(* IEC 61131-3 sources: beckhoffAutomationInterface/ST/Shark/Lib/Sequences, 14 files *)

(* ---- GVL_SequenceConstants.st ---- *)
(* Constants used by Lib/Sequences/* function blocks.
   Lifted from App-side GVL_Constants so Lib code does not depend on
   App-scoped configuration.

   These describe properties of the shared hardware (Bronkhorst PCV needle
   valve) and are identical across all machines that use this valve. *)
{attribute 'qualified_only'}
VAR_GLOBAL CONSTANT
    // Pressure Control Valve (PCV / Needle Valve) Setpoints
    // Bronkhorst Modbus needle valve: 0.0 bar = fully open, 3.0 bar = fully closed
    PCV_CLOSED_SETPOINT : LREAL := 3.0;     // Setpoint that fully closes needle valve (no flow)
    PCV_OPEN_SETPOINT   : LREAL := 0.0;     // Setpoint that fully opens needle valve (max flow)
END_VAR

(* ---- FB_BubblerLeakTestSequence.st ---- *)
(*
FB_BubblerLeakTestSequence
Pressurizes the manifold through a specific bubbler, seals it, and monitors
pressure drop over a configurable test duration.

SEQUENCE:
  1. GasStop:     Ensure both sides shut down
  2. Pressurize:  Fill manifold via MFC + bubbler (CM -> HM path)
  3. Seal:        Close all valves, zero MFC
  4. Stabilize:   Wait for pressure to equalize
  5. Test:        Monitor pressure drop over testDuration
  6. Analyze:     Compare drop vs threshold
  7. Cleanup:     Close all valves
  8. Complete:    Report results

HARDWARE:
  - Side MFC + gas iso valve (carrier gas)
  - CM bubbler valve + CM purge valve (fill path)
  - HM bubbler valve + HM purge valve (propagation to HM)
  - CM/HM pressure sensors (monitor)

OUTPUT:
  - bLeakDetected, fColdManifoldPressureDrop, fHotManifoldPressureDrop
*)
FUNCTION_BLOCK FB_BubblerLeakTestSequence IMPLEMENTS I_TreeNode
VAR
    // Internal State
    _bInitialized    : BOOL := FALSE;
    _bParamsConfigured : BOOL := FALSE;
    _ePhase          : INT := 0;

    // Hardware References
    _ipGasIsoValve        : I_Valve;
    _ipCMBubblerValve     : I_Valve;
    _ipHMBubblerValve     : I_Valve;
    _ipCMPurgeValve       : I_Valve;
    _ipHMPurgeValve       : I_Valve;
    _ipCMVacuumIsoValve   : I_Valve;
    _ipHMVacuumIsoValve   : I_Valve;
    _ipCMPressureSensor   : I_Sensor;
    _ipHMPressureSensor   : I_Sensor;
    _ipMFCController      : I_Controller;

    // Gas stop
    _fbGasStop            : FB_GasStopSequence;

    // Parameters
    _stParams             : ST_CmdBubblerLeakTest;
    _eSide                : E_GasSide;

    // Measurement
    _rCMPressureInitial   : LREAL;
    _rHMPressureInitial   : LREAL;
    _rCMPressureFinal     : LREAL;
    _rHMPressureFinal     : LREAL;

    // Timing
    _fbTimer              : TON;

    // Status
    _bError               : BOOL;
    _sErrorMsg            : STRING(255);
END_VAR

// Output results (readable after completion)
VAR_OUTPUT
    bLeakDetected             : BOOL;
    bColdManifoldLeak         : BOOL;
    bHotManifoldLeak          : BOOL;
    fColdManifoldPressureDrop : LREAL;
    fHotManifoldPressureDrop  : LREAL;
    fPressureDrop             : LREAL;     // max of CM/HM
END_VAR

VAR CONSTANT
    PHASE_IDLE       : INT := 0;
    PHASE_GAS_STOP   : INT := 1;
    PHASE_FILL       : INT := 2;
    PHASE_SEAL       : INT := 3;
    PHASE_STABILIZE  : INT := 4;
    PHASE_TEST       : INT := 5;
    PHASE_ANALYZE    : INT := 6;
    PHASE_CLEANUP    : INT := 7;
    PHASE_DONE       : INT := 8;
    PHASE_ERROR      : INT := 99;
END_VAR

METHOD PUBLIC Init : BOOL
VAR_INPUT
    ipProvider    : I_HardwareProvider;
    eSide         : E_GasSide;
    nBubblerIndex : DINT;
END_VAR
    _bInitialized := FALSE;
    _bParamsConfigured := FALSE;
    _ePhase := PHASE_IDLE;
    _bError := FALSE;
    _sErrorMsg := '';
    _eSide := eSide;

    IF ipProvider = 0 THEN
        GVL_ErrorLogger.Logger.LogError('FB_BubblerLeakTestSequence', E_ErrorId.ERR_GEN_NULL_POINTER, 'Provider is null');
        RETURN;
    END_IF

    IF NOT _fbGasStop.Init(ipProvider := ipProvider, eSide := eSide) THEN RETURN; END_IF

    _ipGasIsoValve := ipProvider.GetGasIsoValve(eSide, nBubblerIndex);
    _ipCMBubblerValve := ipProvider.GetCMBubblerValve(eSide, nBubblerIndex);
    _ipHMBubblerValve := ipProvider.GetHMBubblerValve(eSide, nBubblerIndex);
    _ipCMPurgeValve := ipProvider.GetCMPurgeValve(eSide);
    _ipHMPurgeValve := ipProvider.GetHMPurgeValve(eSide);
    _ipCMVacuumIsoValve := ipProvider.GetCMVacuumIsoValve(eSide);
    _ipHMVacuumIsoValve := ipProvider.GetHMVacuumIsoValve(eSide);
    _ipCMPressureSensor := ipProvider.GetCMPressureSensor(eSide);
    _ipHMPressureSensor := ipProvider.GetHMPressureSensor(eSide);
    _ipMFCController := ipProvider.GetMFCController(eSide);

    IF _ipGasIsoValve = 0 OR _ipCMBubblerValve = 0 OR _ipHMBubblerValve = 0 OR
       _ipCMPurgeValve = 0 OR _ipHMPurgeValve = 0 OR
       _ipCMPressureSensor = 0 OR _ipHMPressureSensor = 0 OR _ipMFCController = 0 THEN
        GVL_ErrorLogger.Logger.LogError('FB_BubblerLeakTestSequence', E_ErrorId.ERR_GEN_NULL_POINTER, 'One or more hardware references are null');
        RETURN;
    END_IF

    _bInitialized := TRUE;
    Init := TRUE;
END_METHOD

METHOD PUBLIC SetParams
VAR_INPUT
    stParams : ST_CmdBubblerLeakTest;
END_VAR
    IF NOT _bInitialized THEN RETURN; END_IF
    _stParams := stParams;
    _bParamsConfigured := TRUE;
END_METHOD

METHOD PUBLIC Tick : ST_NodeResult
VAR
    stResult : ST_NodeResult;
END_VAR
    IF NOT _bInitialized THEN
        Tick.eStatus := E_NodeStatus.FAILURE;
        Tick.bHasError := TRUE;
        Tick.stError.eErrorId := E_ErrorId.ERR_GEN_INITIALIZATION;
        Tick.stError.sSource := 'FB_BubblerLeakTestSequence';
        Tick.stError.sMessage := 'Init must be called before Tick';
        Tick.sDescription := Tick.stError.sMessage;
        RETURN;
    END_IF

    IF NOT _bParamsConfigured THEN
        Tick.eStatus := E_NodeStatus.FAILURE;
        Tick.bHasError := TRUE;
        Tick.stError.eErrorId := E_ErrorId.ERR_GEN_NOT_CONFIGURED;
        Tick.stError.sSource := 'FB_BubblerLeakTestSequence';
        Tick.stError.sMessage := 'SetParams must be called before Tick';
        Tick.sDescription := Tick.stError.sMessage;
        RETURN;
    END_IF

    CASE _ePhase OF
        PHASE_IDLE:
            // Reset outputs
            bLeakDetected := FALSE;
            bColdManifoldLeak := FALSE;
            bHotManifoldLeak := FALSE;
            fColdManifoldPressureDrop := 0.0;
            fHotManifoldPressureDrop := 0.0;
            fPressureDrop := 0.0;
            _fbGasStop.Reset();
            _ePhase := PHASE_GAS_STOP;

        PHASE_GAS_STOP:
            stResult := _fbGasStop.Tick();
            IF stResult.eStatus = E_NodeStatus.SUCCESS THEN
                _ePhase := PHASE_FILL;
                _fbTimer(IN := FALSE);
            ELSIF stResult.eStatus = E_NodeStatus.FAILURE THEN
                _SetError('Gas stop failed');
            END_IF

        PHASE_FILL:
            // Open path: GasIso -> CMBubbler -> CMPurge -> HMPurge -> HMBubbler
            // Set MFC to test flow, wait for fill pressure
            IF NOT _fbTimer.IN THEN
                _ipMFCController.SetSetpoint(REAL_TO_LREAL(_stParams.testFlowRate));
                _ipGasIsoValve.Open();
                _ipCMBubblerValve.Open();
                _ipCMPurgeValve.Open();
                _ipHMPurgeValve.Open();
                _ipHMBubblerValve.Open();
                // Close exhaust paths
                IF _ipCMVacuumIsoValve <> 0 THEN _ipCMVacuumIsoValve.Close(); END_IF
                IF _ipHMVacuumIsoValve <> 0 THEN _ipHMVacuumIsoValve.Close(); END_IF
            END_IF
            _fbTimer(IN := TRUE, PT := DINT_TO_TIME(_stParams.pressureTimeout));
            IF _ipCMPressureSensor.GetMeasurement() >= REAL_TO_LREAL(_stParams.fillPressure) AND
               _ipHMPressureSensor.GetMeasurement() >= REAL_TO_LREAL(_stParams.fillPressure) THEN
                _ePhase := PHASE_SEAL;
                _fbTimer(IN := FALSE);
            ELSIF _fbTimer.Q THEN
                _SetError('Timeout waiting for fill pressure');
            END_IF

        PHASE_SEAL:
            // Close everything, zero MFC
            _ipMFCController.SetSetpoint(0.0);
            _ipGasIsoValve.Close();
            _ipCMBubblerValve.Close();
            _ipHMBubblerValve.Close();
            _ipCMPurgeValve.Close();
            _ipHMPurgeValve.Close();
            _fbTimer(IN := FALSE);
            _ePhase := PHASE_STABILIZE;

        PHASE_STABILIZE:
            _fbTimer(IN := TRUE, PT := DINT_TO_TIME(_stParams.stabilizationTime));
            IF _fbTimer.Q THEN
                // Record initial pressures
                _rCMPressureInitial := _ipCMPressureSensor.GetMeasurement();
                _rHMPressureInitial := _ipHMPressureSensor.GetMeasurement();
                _fbTimer(IN := FALSE);
                _ePhase := PHASE_TEST;
            END_IF

        PHASE_TEST:
            _fbTimer(IN := TRUE, PT := DINT_TO_TIME(_stParams.testDuration));
            IF _fbTimer.Q THEN
                // Record final pressures
                _rCMPressureFinal := _ipCMPressureSensor.GetMeasurement();
                _rHMPressureFinal := _ipHMPressureSensor.GetMeasurement();
                _fbTimer(IN := FALSE);
                _ePhase := PHASE_ANALYZE;
            END_IF

        PHASE_ANALYZE:
            // Calculate pressure drops
            fColdManifoldPressureDrop := _rCMPressureInitial - _rCMPressureFinal;
            fHotManifoldPressureDrop := _rHMPressureInitial - _rHMPressureFinal;

            bColdManifoldLeak := (fColdManifoldPressureDrop > REAL_TO_LREAL(_stParams.leakThreshold));
            bHotManifoldLeak := (fHotManifoldPressureDrop > REAL_TO_LREAL(_stParams.leakThreshold));
            bLeakDetected := bColdManifoldLeak OR bHotManifoldLeak;

            // Max drop for summary
            IF fColdManifoldPressureDrop > fHotManifoldPressureDrop THEN
                fPressureDrop := fColdManifoldPressureDrop;
            ELSE
                fPressureDrop := fHotManifoldPressureDrop;
            END_IF

            _ePhase := PHASE_CLEANUP;

        PHASE_CLEANUP:
            // Ensure all valves closed
            _ipCMBubblerValve.Close();
            _ipHMBubblerValve.Close();
            _ipCMPurgeValve.Close();
            _ipHMPurgeValve.Close();
            _ipGasIsoValve.Close();
            _ePhase := PHASE_DONE;

        PHASE_DONE:
            // Stay done

        PHASE_ERROR:
            // Stay in error
    END_CASE

    IF _ePhase = PHASE_DONE THEN
        Tick.eStatus := E_NodeStatus.SUCCESS;
        Tick.rProgress := 100.0;
        IF bLeakDetected THEN
            Tick.sDescription := CONCAT('LEAK DETECTED - Drop: ', LREAL_TO_STRING(fPressureDrop));
        ELSE
            Tick.sDescription := 'Leak test PASSED';
        END_IF
    ELSIF _ePhase = PHASE_ERROR THEN
        Tick.eStatus := E_NodeStatus.FAILURE;
        Tick.bHasError := TRUE;
        Tick.stError.eErrorId := E_ErrorId.ERR_GEN_INTERNAL;
        Tick.stError.sSource := 'FB_BubblerLeakTestSequence';
        Tick.stError.sMessage := _sErrorMsg;
        Tick.sDescription := _sErrorMsg;
    ELSE
        Tick.eStatus := E_NodeStatus.RUNNING;
        Tick.sDescription := CONCAT('Leak Test: Phase ', INT_TO_STRING(_ePhase));
    END_IF
END_METHOD

METHOD PRIVATE _SetError
VAR_INPUT
    sMsg : STRING(255);
END_VAR
    _sErrorMsg := sMsg;
    _bError := TRUE;
    _ePhase := PHASE_ERROR;
END_METHOD

METHOD PUBLIC Reset : BOOL
    _ePhase := PHASE_IDLE;
    _bError := FALSE;
    _sErrorMsg := '';
    _fbTimer(IN := FALSE);
    bLeakDetected := FALSE;
    bColdManifoldLeak := FALSE;
    bHotManifoldLeak := FALSE;
    fColdManifoldPressureDrop := 0.0;
    fHotManifoldPressureDrop := 0.0;
    fPressureDrop := 0.0;
    _fbGasStop.Reset();
    Reset := TRUE;
END_METHOD

METHOD PUBLIC Halt
    IF _ipMFCController <> 0 THEN _ipMFCController.SetSetpoint(0.0); END_IF
    IF _ipGasIsoValve <> 0 THEN _ipGasIsoValve.Close(); END_IF
    IF _ipCMBubblerValve <> 0 THEN _ipCMBubblerValve.Close(); END_IF
    IF _ipHMBubblerValve <> 0 THEN _ipHMBubblerValve.Close(); END_IF
    IF _ipCMPurgeValve <> 0 THEN _ipCMPurgeValve.Close(); END_IF
    IF _ipHMPurgeValve <> 0 THEN _ipHMPurgeValve.Close(); END_IF
    Reset();
END_METHOD

PROPERTY PUBLIC NodeName : STRING(50)
    GET
        NodeName := 'BubblerLeakTest';
    END_GET
END_PROPERTY

END_FUNCTION_BLOCK

(* ---- FB_BubblerPurgeSequence.st ---- *)
(*
FB_BubblerPurgeSequence
Purge a specific bubbler: Prepare exhaust -> CM purge -> delay -> HM purge.
*)
FUNCTION_BLOCK FB_BubblerPurgeSequence IMPLEMENTS I_TreeNode
VAR
    _seq : FB_SequenceNode;
    // Steps
    stepPrepareExhaust : FB_PrepareExhaustSequence;
    stepBubblerPurgeCM : FB_BubblerPurgeCMSequence;
    stepDelay          : FB_WaitNode;
    stepBubblerPurgeHM : FB_BubblerPurgeHMSequence;

    // Internal state
    _bInitialized    : BOOL := FALSE;
    _eSide           : E_GasSide;
    _nBubblerIndex   : DINT;
END_VAR

VAR CONSTANT
    SWITCH_DELAY : TIME := T#2S;
END_VAR

METHOD PUBLIC Init : BOOL
VAR_INPUT
    ipProvider    : I_HardwareProvider;
    eSide         : E_GasSide;
    nBubblerIndex : DINT;
END_VAR
    IF _bInitialized THEN
        IF _eSide = eSide AND _nBubblerIndex = nBubblerIndex THEN
            Init := TRUE;
            RETURN;
        END_IF
        _seq.ClearChildren();
        _bInitialized := FALSE;
    END_IF

    IF ipProvider = 0 THEN
        GVL_ErrorLogger.Logger.LogError('FB_BubblerPurgeSequence', E_ErrorId.ERR_GEN_NULL_POINTER, 'Provider is null');
        RETURN;
    END_IF
    _eSide := eSide;
    _nBubblerIndex := nBubblerIndex;

    stepPrepareExhaust.Init(ipProvider, eSide);
    stepPrepareExhaust.NodeName := 'PrepareExhaust';
    _seq.AddChild(stepPrepareExhaust);

    stepBubblerPurgeCM.Init(ipProvider, eSide, nBubblerIndex);
    stepBubblerPurgeCM.NodeName := 'BubblerPurgeCM';
    _seq.AddChild(stepBubblerPurgeCM);

    stepDelay.Init(tWaitTime := SWITCH_DELAY, sNodeName := 'SwitchDelay');
    _seq.AddChild(stepDelay);

    stepBubblerPurgeHM.Init(ipProvider, eSide, nBubblerIndex);
    stepBubblerPurgeHM.NodeName := 'BubblerPurgeHM';
    _seq.AddChild(stepBubblerPurgeHM);

    _seq.sName := CONCAT(CONCAT('BubblerPurgeFull_Side', TO_STRING(eSide)), CONCAT('_Idx', TO_STRING(nBubblerIndex)));

    _bInitialized := TRUE;
    Init := TRUE;
END_METHOD

METHOD PUBLIC SetParams
VAR_INPUT
    stCmd : ST_CmdPurge;
END_VAR
    IF NOT _bInitialized THEN RETURN; END_IF

    stepBubblerPurgeCM.SetParams(
        nPurgeCycles           := stCmd.coldManifoldPurgeCycles,
        rPurgeFlowRate         := REAL_TO_LREAL(stCmd.purgeGasFlow),
        rPurgePressure         := REAL_TO_LREAL(stCmd.purgeHighPressureLimit),
        rEvacuationPressure    := REAL_TO_LREAL(stCmd.purgeLowPressureLimit),
        tPressurizationTimeout := DINT_TO_TIME(stCmd.highPressureTimeout),
        tEvacuationTimeout     := DINT_TO_TIME(stCmd.lowPressureTimeout)
    );

    stepBubblerPurgeHM.SetParams(
        nPurgeCycles           := stCmd.hotManifoldPurgeCycles,
        rPurgeFlowRate         := REAL_TO_LREAL(stCmd.purgeGasFlow),
        rPurgePressure         := REAL_TO_LREAL(stCmd.purgeHighPressureLimit),
        rFinalPressure         := REAL_TO_LREAL(stCmd.hotManifoldOperatingPressure),
        rEvacuationPressure    := REAL_TO_LREAL(stCmd.purgeLowPressureLimit),
        tPressurizationTimeout := DINT_TO_TIME(stCmd.highPressureTimeout),
        tEvacuationTimeout     := DINT_TO_TIME(stCmd.lowPressureTimeout)
    );
END_METHOD

PROPERTY PUBLIC NodeName : STRING(50)
    GET
        NodeName := _seq.sName;
    END_GET
    SET
        _seq.sName := NodeName;
    END_SET
END_PROPERTY

METHOD Tick : ST_NodeResult
    IF NOT _bInitialized THEN
        Tick.eStatus := E_NodeStatus.FAILURE;
        Tick.bHasError := TRUE;
        Tick.stError.eErrorId := E_ErrorId.ERR_GEN_INITIALIZATION;
        Tick.stError.sSource := 'FB_BubblerPurgeSequence';
        Tick.stError.sMessage := 'Init must be called before Tick';
        Tick.sDescription := Tick.stError.sMessage;
        RETURN;
    END_IF

    Tick := _seq.Tick();
END_METHOD

{attribute 'estimated-stack-usage' := '500'}
METHOD Reset : BOOL
    Reset := _seq.Reset();
END_METHOD

{attribute 'estimated-stack-usage' := '500'}
METHOD Halt
    _seq.Halt();
END_METHOD

END_FUNCTION_BLOCK

(* ---- FB_ChuckVacuumHoldSequence.st ---- *)
// FB_ChuckVacuumHoldSequence (Lib)
//
// Machine-agnostic chuck-vacuum hold sequence. All hardware-specific
// behavior (pump topology, vent valve presence, sensor type) is delegated
// to the machine-specific I_ChuckVacuumSystem implementation provided by
// the hardware provider.
//
// SEQUENCE:
//   Idle           -> PrepareForHold() then wait pump stabilize
//   VerifyingPump  -> after stabilize, open zone valves
//   OpeningValves  -> hierarchical open 1..nZoneCount, then watch sensor
//   WaitingVacuum  -> until IsVacuumHeld OR timeout
//   Done / Error
FUNCTION_BLOCK FB_ChuckVacuumHoldSequence IMPLEMENTS I_TreeNode
VAR
    _bInitialized    : BOOL := FALSE;
    _eState          : E_ChuckVacuumState := E_ChuckVacuumState.Idle;

    _ipChuckVacuum   : I_ChuckVacuumSystem;

    // Parameters
    _nZoneCount              : INT  := 1;
    _tTimeout                : TIME := T#1M;
    _rLockPressureThreshold  : LREAL := 0.65;

    _fbTimer         : TON;
    _bError          : BOOL;
    _sErrorMsg       : STRING(255);
END_VAR

VAR CONSTANT
    PUMP_STABILIZE_TIME : TIME := T#500MS;
END_VAR

METHOD PUBLIC Init : BOOL
VAR_INPUT
    ipProvider : I_HardwareProvider;
END_VAR
    _bInitialized := FALSE;
    _eState := E_ChuckVacuumState.Idle;
    _bError := FALSE;
    _sErrorMsg := '';

    IF ipProvider = 0 THEN
        GVL_ErrorLogger.Logger.LogError('FB_ChuckVacuumHoldSequence', E_ErrorId.ERR_GEN_NULL_POINTER, 'Provider is null');
        RETURN;
    END_IF

    _ipChuckVacuum := ipProvider.GetChuckVacuumSystem();
    IF _ipChuckVacuum = 0 THEN
        GVL_ErrorLogger.Logger.LogError('FB_ChuckVacuumHoldSequence', E_ErrorId.ERR_GEN_NULL_POINTER, 'Chuck vacuum subsystem not available');
        RETURN;
    END_IF

    IF NOT _ipChuckVacuum.IsInitialized() THEN
        GVL_ErrorLogger.Logger.LogError('FB_ChuckVacuumHoldSequence', E_ErrorId.ERR_GEN_NULL_POINTER, 'Chuck vacuum subsystem not initialized');
        RETURN;
    END_IF

    _bInitialized := TRUE;
    Init := TRUE;
END_METHOD

METHOD PUBLIC SetParams
VAR_INPUT
    stParams : ST_ChuckVacuumHold;
END_VAR
VAR
    nMax : INT;
END_VAR
    IF NOT _bInitialized THEN RETURN; END_IF
    nMax := _ipChuckVacuum.GetMaxZoneCount();
    _nZoneCount := LIMIT(1, stParams.iSelectZone, nMax);
    _tTimeout := stParams.tPressureTimeout;
    _rLockPressureThreshold := REAL_TO_LREAL(stParams.fLockPressureThreshold);
END_METHOD

METHOD PUBLIC Tick : ST_NodeResult
VAR
    i : INT;
END_VAR
    IF NOT _bInitialized THEN
        _sErrorMsg := 'Init must be called before Tick';
        _bError := TRUE;
        _eState := E_ChuckVacuumState.Error;
        Tick.eStatus := E_NodeStatus.FAILURE;
        Tick.bHasError := TRUE;
        Tick.stError.eErrorId := E_ErrorId.ERR_GEN_INITIALIZATION;
        Tick.stError.sSource := 'FB_ChuckVacuumHoldSequence';
        Tick.stError.sMessage := _sErrorMsg;
        Tick.sDescription := _sErrorMsg;
        RETURN;
    END_IF

    CASE _eState OF
        E_ChuckVacuumState.Idle:
            // Close vent (if any), ensure pump source is active
            _ipChuckVacuum.PrepareForHold();
            _eState := E_ChuckVacuumState.VerifyingPump;
            _fbTimer(IN := FALSE);

        E_ChuckVacuumState.VerifyingPump:
            // Brief stabilization window for pump/vent valve to settle
            _fbTimer(IN := TRUE, PT := PUMP_STABILIZE_TIME);
            IF _fbTimer.Q THEN
                _fbTimer(IN := FALSE);
                _eState := E_ChuckVacuumState.OpeningValves;
            END_IF

        E_ChuckVacuumState.OpeningValves:
            // Open zone valves hierarchically (innermost first)
            FOR i := 1 TO _nZoneCount DO
                _ipChuckVacuum.OpenZone(nZone := i);
            END_FOR
            _eState := E_ChuckVacuumState.WaitingVacuum;
            _fbTimer(IN := FALSE);

        E_ChuckVacuumState.WaitingVacuum:
            _fbTimer(IN := TRUE, PT := _tTimeout);
            IF _fbTimer.Q THEN
                _sErrorMsg := 'Timeout waiting for vacuum';
                _bError := TRUE;
                _eState := E_ChuckVacuumState.Error;
            ELSIF _ipChuckVacuum.IsVacuumHeld(nActiveZoneCount := _nZoneCount, rThreshold := _rLockPressureThreshold) THEN
                _eState := E_ChuckVacuumState.Done;
            END_IF

        E_ChuckVacuumState.Done:
            ; // terminal
        E_ChuckVacuumState.Error:
            ; // terminal until Reset
    END_CASE

    Tick.eStatus := E_NodeStatus.RUNNING;
    Tick.rProgress := 0.0;
    Tick.bHasError := _bError;
    Tick.sDescription := 'Applying Vacuum';

    IF _eState = E_ChuckVacuumState.Done THEN
        Tick.eStatus := E_NodeStatus.SUCCESS;
        Tick.rProgress := 100.0;
        Tick.sDescription := 'Vacuum Held';
    ELSIF _eState = E_ChuckVacuumState.Error THEN
        Tick.eStatus := E_NodeStatus.FAILURE;
        Tick.bHasError := TRUE;
        Tick.stError.eErrorId := E_ErrorId.ERR_GEN_TIMEOUT;
        Tick.stError.sSource := 'FB_ChuckVacuumHoldSequence';
        Tick.stError.sMessage := _sErrorMsg;
        Tick.stError.fExpectedValue := TO_REAL(_rLockPressureThreshold);
        Tick.stError.sUnits := 'bar';
        Tick.sDescription := _sErrorMsg;
    END_IF
END_METHOD

METHOD PUBLIC GetState : E_ChuckVacuumState
    GetState := _eState;
END_METHOD

METHOD PUBLIC Reset : BOOL
    _eState := E_ChuckVacuumState.Idle;
    _bError := FALSE;
    _sErrorMsg := '';
    _fbTimer(IN := FALSE);
    IF _ipChuckVacuum <> 0 THEN
        _ipChuckVacuum.Reset();
    END_IF
    Reset := TRUE;
END_METHOD

METHOD PUBLIC Halt
    Reset();
END_METHOD

END_FUNCTION_BLOCK

(* ---- FB_ChuckVacuumReleaseSequence.st ---- *)
// FB_ChuckVacuumReleaseSequence (Lib)
//
// Machine-agnostic chuck-vacuum release sequence. All hardware-specific
// behavior is delegated to the I_ChuckVacuumSystem implementation.
//
// SEQUENCE:
//   Idle           -> close all zones, BeginRelease()  (opens vent if any)
//   WaitingVacuum  -> until IsVacuumReleased OR timeout
//   On release    -> FinishRelease() (stops pump if dedicated)
//   Done / Error
FUNCTION_BLOCK FB_ChuckVacuumReleaseSequence IMPLEMENTS I_TreeNode
VAR
    _bInitialized    : BOOL := FALSE;
    _eState          : E_ChuckVacuumState := E_ChuckVacuumState.Idle;

    _ipChuckVacuum   : I_ChuckVacuumSystem;

    // Parameters
    _tTimeout                   : TIME  := T#1M;
    _rReleasePressureThreshold  : LREAL := 0.8;

    _fbTimer         : TON;
    _bError          : BOOL;
    _sErrorMsg       : STRING(255);
END_VAR

METHOD PUBLIC Init : BOOL
VAR_INPUT
    ipProvider : I_HardwareProvider;
END_VAR
    _bInitialized := FALSE;
    _eState := E_ChuckVacuumState.Idle;
    _bError := FALSE;
    _sErrorMsg := '';

    IF ipProvider = 0 THEN
        GVL_ErrorLogger.Logger.LogError('FB_ChuckVacuumReleaseSequence', E_ErrorId.ERR_GEN_NULL_POINTER, 'Provider is null');
        RETURN;
    END_IF

    _ipChuckVacuum := ipProvider.GetChuckVacuumSystem();
    IF _ipChuckVacuum = 0 THEN
        GVL_ErrorLogger.Logger.LogError('FB_ChuckVacuumReleaseSequence', E_ErrorId.ERR_GEN_NULL_POINTER, 'Chuck vacuum subsystem not available');
        RETURN;
    END_IF

    IF NOT _ipChuckVacuum.IsInitialized() THEN
        GVL_ErrorLogger.Logger.LogError('FB_ChuckVacuumReleaseSequence', E_ErrorId.ERR_GEN_NULL_POINTER, 'Chuck vacuum subsystem not initialized');
        RETURN;
    END_IF

    _bInitialized := TRUE;
    Init := TRUE;
END_METHOD

METHOD PUBLIC SetParams
VAR_INPUT
    stParams : ST_ChuckVacuumRelease;
END_VAR
    IF NOT _bInitialized THEN RETURN; END_IF
    _tTimeout := stParams.tPressureTimeout;
    _rReleasePressureThreshold := REAL_TO_LREAL(stParams.fReleasePressureThreshold);
END_METHOD

METHOD PUBLIC Tick : ST_NodeResult
VAR
    i, nMax : INT;
END_VAR
    IF NOT _bInitialized THEN
        _sErrorMsg := 'Init must be called before Tick';
        _bError := TRUE;
        _eState := E_ChuckVacuumState.Error;
        Tick.eStatus := E_NodeStatus.FAILURE;
        Tick.bHasError := TRUE;
        Tick.stError.eErrorId := E_ErrorId.ERR_GEN_INITIALIZATION;
        Tick.stError.sSource := 'FB_ChuckVacuumReleaseSequence';
        Tick.stError.sMessage := _sErrorMsg;
        Tick.sDescription := _sErrorMsg;
        RETURN;
    END_IF

    CASE _eState OF
        E_ChuckVacuumState.Idle:
            _eState := E_ChuckVacuumState.OpeningValves;
            _fbTimer(IN := FALSE);

        E_ChuckVacuumState.OpeningValves:
            // Close every zone, then open vent (if any) via BeginRelease
            nMax := _ipChuckVacuum.GetMaxZoneCount();
            FOR i := 1 TO nMax DO
                _ipChuckVacuum.CloseZone(nZone := i);
            END_FOR
            _ipChuckVacuum.BeginRelease();
            _eState := E_ChuckVacuumState.WaitingVacuum;
            _fbTimer(IN := FALSE);

        E_ChuckVacuumState.WaitingVacuum:
            _fbTimer(IN := TRUE, PT := _tTimeout);
            IF _fbTimer.Q THEN
                _sErrorMsg := 'Timeout waiting for vacuum release';
                _bError := TRUE;
                _eState := E_ChuckVacuumState.Error;
            ELSIF _ipChuckVacuum.IsVacuumReleased(rThreshold := _rReleasePressureThreshold) THEN
                // Stop pump (no-op when pump is shared)
                _ipChuckVacuum.FinishRelease();
                _eState := E_ChuckVacuumState.Done;
            END_IF

        E_ChuckVacuumState.Done:
            ; // terminal
        E_ChuckVacuumState.Error:
            ; // terminal until Reset
    END_CASE

    Tick.eStatus := E_NodeStatus.RUNNING;
    Tick.rProgress := 0.0;
    Tick.bHasError := _bError;
    Tick.sDescription := 'Releasing Vacuum';

    IF _eState = E_ChuckVacuumState.Done THEN
        Tick.eStatus := E_NodeStatus.SUCCESS;
        Tick.rProgress := 100.0;
        Tick.sDescription := 'Vacuum Released';
    ELSIF _eState = E_ChuckVacuumState.Error THEN
        Tick.eStatus := E_NodeStatus.FAILURE;
        Tick.bHasError := TRUE;
        Tick.stError.eErrorId := E_ErrorId.ERR_GEN_TIMEOUT;
        Tick.stError.sSource := 'FB_ChuckVacuumReleaseSequence';
        Tick.stError.sMessage := _sErrorMsg;
        Tick.stError.fExpectedValue := TO_REAL(_rReleasePressureThreshold);
        Tick.stError.sUnits := 'bar';
        Tick.sDescription := _sErrorMsg;
    END_IF
END_METHOD

METHOD PUBLIC GetState : E_ChuckVacuumState
    GetState := _eState;
END_METHOD

METHOD PUBLIC Reset : BOOL
    _eState := E_ChuckVacuumState.Idle;
    _bError := FALSE;
    _sErrorMsg := '';
    _fbTimer(IN := FALSE);
    IF _ipChuckVacuum <> 0 THEN
        _ipChuckVacuum.Reset();
    END_IF
    Reset := TRUE;
END_METHOD

METHOD PUBLIC Halt
    Reset();
END_METHOD

END_FUNCTION_BLOCK

(* ---- FB_GasStartSequence.st ---- *)
(*
FB_GasStartSequence — Starts bubbler flow for one side.

  ── Refactor of FB_GasStartSequence: "lazy build" architecture ──
  The original built the tree in Init() with placeholder 0.0 values for every
  parameter-driven step, then overwrote them in SetParams() via property setters.
  That split made Init() ambiguous (is a 0.0 real or a placeholder?) and left
  the I14 risk that a skipped SetParams leaves waits with target 0.0.

  This version separates the two kinds of configuration cleanly:
    Init()       → resolve + validate HARDWARE only. No tree, no setpoints.
    SetParams()  → validate params, DERIVE every runtime value, then _BuildTree().
    _BuildTree() → the single recipe: wire each node ONCE with its final value.

  Result: no placeholders anywhere; reading _BuildTree() shows every real value.

Physical path:
  Gas Inlet (3 bar ± 0.5) → MFC → CM [sensor] → CM bubbler valve → Bubbler (heated) →
  HM bubbler valve → HM [sensor] → PCV → Start valve → Micro nozzle → Reactor (~1 bar)

Terminology:
  CM (Cold Manifold) = "distributor" side — MFC feeds here; CM sensor reads here.
  HM (Hot Manifold) = "combiner" side  — after bubbler; PCV controls pressure here.

Phases:
  0. Open PCV fully        : allow free flow during evacuation
  1. Evacuate HM           : open exhaust iso + HM vacuum iso; wait HM < 0.5 bar;
                             close HM vacuum iso
  2. Fill via purge valves : MFC max flow + gas inlet + HM/CM purge open;
                             wait CM > 2.0 bar; close purge valves; stop MFC + close gas inlet
  3. Path-open check       : open start valve + HM bubbler; wait HM < 1.3 bar;
                             close start valve
  4. Establish flow        : reopen start valve; restart MFC + gas inlet;
                             wait CM > CM operating target; wait HM < HM operating target;
                             open CM bubbler; wait HM within tolerance of target;
                             set final MFC flow rate
*)
FUNCTION_BLOCK FB_GasStartSequence IMPLEMENTS I_TreeNode
VAR
    _seq : FB_SequenceNode;

    // Phase 0: Open PCV fully to allow free flow during evacuation
    stepOpenPCVFully      : FB_SetControllerNode;

    // Phase 1: Unconditional evacuation via exhaust pump + HM vacuum iso
    stepOpenExhaustPump   : FB_OpenValveNode;     // Open main exhaust iso valve (VALV_EX_PUMP)
    stepOpenHMVacuumIso   : FB_OpenValveNode;     // Open HM vacuum iso (connects HM to exhaust path)
    stepWaitEvacuation    : FB_WaitForSensorNode; // Wait HM < MIN_EVACUATION_PRESSURE (PCV stays fully open)
    stepCloseHMVacuumIso  : FB_CloseValveNode;    // Close HM vacuum iso

    // Phase 2: Fill manifolds through purge valves with max MFC flow
    stepSetMFCBuildupFlow : FB_SetControllerNode; // MFC = _rBuildupFlow
    stepOpenGasInlet      : FB_OpenValveNode;     // Open gas iso valve
    stepOpenHMPurge       : FB_OpenValveNode;     // Open HM purge valve
    stepOpenCMPurge       : FB_OpenValveNode;     // Open CM purge valve
    stepWaitCMFilled      : FB_WaitForSensorNode; // Wait CM > CM_FILL_PRESSURE (2.0 bar)
    stepCloseHMPurge      : FB_CloseValveNode;    // Close HM purge valve
    stepCloseCMPurge      : FB_CloseValveNode;    // Close CM purge valve
    stepStopMFC           : FB_SetControllerNode; // MFC = 0 (stop flow)
    stepCloseGasInlet     : FB_CloseValveNode;    // Close gas iso valve

    // Phase 3: Path-open check — connect HM to reactor side; verify HM near atmospheric
    stepOpenStartValve1   : FB_OpenValveNode;     // Open start (nozzle iso) valve
    stepOpenHMBubbler     : FB_OpenValveNode;     // Open HM bubbler valve
    stepWaitHMPressureDown: FB_WaitForSensorNode; // Wait HM < HM_ATMOS_CHECK_PRESSURE (1.3 bar)
    stepCloseStartValve   : FB_CloseValveNode;    // Close start valve (re-isolate for Phase 4 fill)

    // Phase 4: Establish operating flow
    stepOpenStartValve2   : FB_OpenValveNode;     // Re-open start valve
    stepSetMFCBuildupFlow2: FB_SetControllerNode; // MFC = _rBuildupFlow (second time)
    stepOpenGasInlet2     : FB_OpenValveNode;     // Re-open gas inlet (second time)
    stepWaitCMAtTarget    : FB_WaitForSensorNode; // Wait CM > _rCMAtTarget (CM operating pressure)
    stepSetPCVOperating   : FB_SetControllerNode; // Set PCV = _rHMTarget — engage back-pressure control
    stepWaitHMBelowTarget : FB_WaitForSensorNode; // Wait HM < _rHMTarget (HM operating pressure)
    stepOpenCMBubbler     : FB_OpenValveNode;     // Open CM bubbler valve
    stepWaitHMAtTarget    : FB_WaitForSensorNode; // Wait HM within _rHMTolerance of _rHMTarget
    stepSetMFCTarget      : FB_SetControllerNode; // MFC = _rFinalFlow (final target flow)

    // ── Hardware references (resolved in Init) ──
    _ipGasIsoValve           : I_Valve;
    _ipCMBubblerValve        : I_Valve;
    _ipHMBubblerValve        : I_Valve;
    _ipHMPurgeValve          : I_Valve;
    _ipCMPurgeValve          : I_Valve;
    _ipHMVacuumIsoValve      : I_Valve;
    _ipNozzleIsoValve        : I_Valve;
    _ipCMPressureSensor      : I_Sensor;
    _ipHMPressureSensor      : I_Sensor;
    _ipMFCController         : I_Controller;
    _ipPressureController    : I_Controller;
    _ipExhaustVacuumIsoValve : I_Valve;

    // ── Init-scoped config ──
    _tEvacuationTimeout : TIME;

    // ── Runtime values (derived in SetParams; consumed by _BuildTree) ──
    _rBuildupFlow       : LREAL;   // MFC buildup/purge flow
    _rCMAtTarget        : LREAL;   // CM operating target = HM target + gradient margin
    _rHMTarget          : LREAL;   // HM operating pressure (PCV setpoint + HM waits)
    _rHMTolerance       : LREAL;   // HM in-range tolerance band (bar)
    _rFinalFlow         : LREAL;   // Final operating MFC flow rate
    _tCMPressureTimeout : TIME;    // CM wait timeout
    _tHMPressureTimeout : TIME;    // HM wait timeout

    // Internal state
    _bInitialized      : BOOL := FALSE;
    _bParamsConfigured : BOOL := FALSE;
    _eSide             : E_GasSide;
    _nBubblerIndex     : DINT;
END_VAR

VAR CONSTANT
    MIN_EVACUATION_PRESSURE   : LREAL := 0.5;   // Bar — HM evacuation wait target
    CM_FILL_PRESSURE          : LREAL := 2.0;   // Bar — CM fill target via purge valves
    MAX_BUILDUP_FLOW_RATE     : LREAL := 23.0;  // sccm — MFC flow for manifold fill/purge
    HM_ATMOS_CHECK_PRESSURE   : LREAL := 1.3;   // Bar — HM target for path-open check (near atmospheric)
    GRADIENT_MARGIN           : LREAL := 0.2;   // Bar — CM must lead HM by this for forward flow
    HEAD_OPERATING_PRESSURE   : LREAL := 1.0;   // Bar — reactor head steady-state pressure
    MIN_PRESSURE_DIFFERENTIAL : LREAL := 0.2;   // Bar — minimum HM-to-head differential for flow
END_VAR

(* Init — resolve and validate hardware ONLY. Does not build the tree.
   The tree is built by SetParams() once every runtime value is known. *)
METHOD PUBLIC Init : BOOL
VAR_INPUT
    ipProvider         : I_HardwareProvider;
    eSide              : E_GasSide;
    nBubblerIndex      : DINT := 1;
    tEvacuationTimeout : TIME := T#30S;
END_VAR
    // Re-init guard: same side/index → no-op; different → drop any prior build
    IF _bInitialized THEN
        IF _eSide = eSide AND _nBubblerIndex = nBubblerIndex THEN
            Init := TRUE;
            RETURN;
        END_IF
        _seq.ClearChildren();
        _bInitialized := FALSE;
        _bParamsConfigured := FALSE;
    END_IF

    IF ipProvider = 0 THEN
        GVL_ErrorLogger.Logger.LogError('FB_GasStartSequence', E_ErrorId.ERR_GEN_NULL_POINTER, 'Provider is null');
        RETURN;
    END_IF

    _eSide := eSide;
    _nBubblerIndex := nBubblerIndex;
    _tEvacuationTimeout := tEvacuationTimeout;

    // Resolve hardware references into members
    _ipGasIsoValve           := ipProvider.GetGasIsoValve(eSide, nBubblerIndex);
    _ipCMBubblerValve        := ipProvider.GetCMBubblerValve(eSide, nBubblerIndex);
    _ipHMBubblerValve        := ipProvider.GetHMBubblerValve(eSide, nBubblerIndex);
    _ipHMPurgeValve          := ipProvider.GetHMPurgeValve(eSide);
    _ipCMPurgeValve          := ipProvider.GetCMPurgeValve(eSide);
    _ipHMVacuumIsoValve      := ipProvider.GetHMVacuumIsoValve(eSide);
    _ipNozzleIsoValve        := ipProvider.GetNozzleIsoValve(eSide);
    _ipCMPressureSensor      := ipProvider.GetCMPressureSensor(eSide);
    _ipHMPressureSensor      := ipProvider.GetHMPressureSensor(eSide);
    _ipMFCController         := ipProvider.GetMFCController(eSide);
    _ipPressureController    := ipProvider.GetPressureController(eSide);
    _ipExhaustVacuumIsoValve := ipProvider.GetExhaustVacuumIsoValve();

    // Validate all hardware
    IF _ipGasIsoValve = 0 OR _ipCMBubblerValve = 0 OR _ipHMBubblerValve = 0 OR
       _ipHMPurgeValve = 0 OR _ipCMPurgeValve = 0 OR _ipHMVacuumIsoValve = 0 OR
       _ipNozzleIsoValve = 0 OR _ipCMPressureSensor = 0 OR _ipHMPressureSensor = 0 OR
       _ipMFCController = 0 OR _ipPressureController = 0 OR _ipExhaustVacuumIsoValve = 0 THEN
        GVL_ErrorLogger.Logger.LogError('FB_GasStartSequence', E_ErrorId.ERR_GEN_NULL_POINTER, 'One or more hardware references are null');
        RETURN;
    END_IF

    _seq.sName := CONCAT(CONCAT('GasStart_', TO_STRING(eSide)), CONCAT('_Idx', TO_STRING(nBubblerIndex)));
    _bParamsConfigured := FALSE;
    _bInitialized := TRUE;
    Init := TRUE;
END_METHOD

(* SetParams — validate the command, derive every runtime value, then build the tree.
   After this returns TRUE, no node holds a placeholder value. *)
METHOD PUBLIC SetParams : BOOL
VAR_INPUT
    stParams : ST_CmdStartBubblerFlow;
END_VAR
VAR
    rHMTarget      : LREAL;
    rFlowTolerance : LREAL;
END_VAR
    IF NOT _bInitialized THEN RETURN; END_IF

    rHMTarget := REAL_TO_LREAL(stParams.hotManifoldOperatingPressure);

    // Validate: pressure differential must be sufficient for flow
    IF (rHMTarget - HEAD_OPERATING_PRESSURE) < MIN_PRESSURE_DIFFERENTIAL THEN
        GVL_ErrorLogger.Logger.LogError(
            'FB_GasStartSequence',
            E_ErrorId.ERR_GEN_INVALID_PARAM,
            'hotManifoldOperatingPressure too low — insufficient pressure differential for flow');
        RETURN;
    END_IF

    IF REAL_TO_LREAL(stParams.flowRate) <= 0.0 THEN
        GVL_ErrorLogger.Logger.LogError(
            'FB_GasStartSequence',
            E_ErrorId.ERR_GEN_INVALID_PARAM,
            'flowRate must be > 0');
        RETURN;
    END_IF

    rFlowTolerance := REAL_TO_LREAL(stParams.MFCFlowRateTolerance);

    // ── Derive every runtime value here (single place; no placeholders) ──
    _rHMTarget          := rHMTarget;
    _rBuildupFlow       := MAX(REAL_TO_LREAL(stParams.flowRate), MAX_BUILDUP_FLOW_RATE);
    _rCMAtTarget        := rHMTarget + GRADIENT_MARGIN;   // CM must lead HM for forward flow
    _rHMTolerance       := rHMTarget * (rFlowTolerance / 100.0);
    _rFinalFlow         := REAL_TO_LREAL(stParams.flowRate);
    _tCMPressureTimeout := DINT_TO_TIME(REAL_TO_DINT(stParams.coldManifoldPressureTimeout));
    _tHMPressureTimeout := DINT_TO_TIME(REAL_TO_DINT(stParams.hotManifoldPressureTimeout));

    // Build (or rebuild) the tree now that every value is final
    _seq.ClearChildren();
    _BuildTree();

    _bParamsConfigured := TRUE;
    SetParams := TRUE;
END_METHOD

(* _BuildTree — the single recipe. Every node is wired ONCE with its final value:
   constants for fixed steps, derived members _r*/_t* for parameter-driven steps. *)
METHOD PRIVATE _BuildTree
    // Phase 0 — Open PCV fully to allow free flow during evacuation.
    stepOpenPCVFully.Init(ipController := _ipPressureController, rSetpoint := GVL_SequenceConstants.PCV_OPEN_SETPOINT, sNodeName := 'OpenPCVFully');
    _seq.AddChild(stepOpenPCVFully);

    // Phase 1 — Unconditional evacuation via exhaust pump + HM vacuum iso.
    stepOpenExhaustPump.Init(ipValve := _ipExhaustVacuumIsoValve, sNodeName := 'OpenExhaustPump');
    _seq.AddChild(stepOpenExhaustPump);

    stepOpenHMVacuumIso.Init(ipValve := _ipHMVacuumIsoValve, sNodeName := 'OpenHMVacuumIso');
    _seq.AddChild(stepOpenHMVacuumIso);

    stepWaitEvacuation.Init(ipSensor := _ipHMPressureSensor, rTarget := MIN_EVACUATION_PRESSURE, eMode := E_CompareMode.LESS_THAN, tTimeout := _tEvacuationTimeout, sNodeName := 'WaitEvacuation');
    _seq.AddChild(stepWaitEvacuation);

    stepCloseHMVacuumIso.Init(ipValve := _ipHMVacuumIsoValve, sNodeName := 'CloseHMVacuumIso');
    _seq.AddChild(stepCloseHMVacuumIso);

    // Phase 2 — Fill manifolds through purge valves; wait CM fills to 2.0 bar.
    stepSetMFCBuildupFlow.Init(ipController := _ipMFCController, rSetpoint := _rBuildupFlow, sNodeName := 'SetMFCBuildup');
    _seq.AddChild(stepSetMFCBuildupFlow);

    stepOpenGasInlet.Init(ipValve := _ipGasIsoValve, sNodeName := 'OpenGasInlet');
    _seq.AddChild(stepOpenGasInlet);

    stepOpenHMPurge.Init(ipValve := _ipHMPurgeValve, sNodeName := 'OpenHMPurge');
    _seq.AddChild(stepOpenHMPurge);

    stepOpenCMPurge.Init(ipValve := _ipCMPurgeValve, sNodeName := 'OpenCMPurge');
    _seq.AddChild(stepOpenCMPurge);

    stepWaitCMFilled.Init(ipSensor := _ipCMPressureSensor, rTarget := CM_FILL_PRESSURE, eMode := E_CompareMode.GREATER_THAN, tTimeout := _tCMPressureTimeout, sNodeName := 'WaitCMFilled');
    _seq.AddChild(stepWaitCMFilled);

    stepCloseHMPurge.Init(ipValve := _ipHMPurgeValve, sNodeName := 'CloseHMPurge');
    _seq.AddChild(stepCloseHMPurge);

    stepCloseCMPurge.Init(ipValve := _ipCMPurgeValve, sNodeName := 'CloseCMPurge');
    _seq.AddChild(stepCloseCMPurge);

    stepStopMFC.Init(ipController := _ipMFCController, rSetpoint := 0.0, sNodeName := 'StopMFC');
    _seq.AddChild(stepStopMFC);

    // Phase 3 — Path-open check: connect HM to reactor; verify HM near atmospheric.
    stepOpenStartValve1.Init(ipValve := _ipNozzleIsoValve, sNodeName := 'OpenStartValve1');
    _seq.AddChild(stepOpenStartValve1);

    stepOpenHMBubbler.Init(ipValve := _ipHMBubblerValve, sNodeName := 'OpenHMBubbler');
    _seq.AddChild(stepOpenHMBubbler);

    stepWaitHMPressureDown.Init(ipSensor := _ipHMPressureSensor, rTarget := HM_ATMOS_CHECK_PRESSURE, eMode := E_CompareMode.LESS_THAN, tTimeout := _tHMPressureTimeout, sNodeName := 'WaitHMPressureDown');
    _seq.AddChild(stepWaitHMPressureDown);

    stepCloseStartValve.Init(ipValve := _ipNozzleIsoValve, sNodeName := 'CloseStartValve');
    _seq.AddChild(stepCloseStartValve);

    // Phase 4 — Establish operating flow.
    stepOpenStartValve2.Init(ipValve := _ipNozzleIsoValve, sNodeName := 'OpenStartValve2');
    _seq.AddChild(stepOpenStartValve2);

    stepSetMFCBuildupFlow2.Init(ipController := _ipMFCController, rSetpoint := _rBuildupFlow, sNodeName := 'SetMFCBuildup2');
    _seq.AddChild(stepSetMFCBuildupFlow2);

    stepOpenGasInlet2.Init(ipValve := _ipGasIsoValve, sNodeName := 'OpenGasInlet2');
    _seq.AddChild(stepOpenGasInlet2);

    stepWaitCMAtTarget.Init(ipSensor := _ipCMPressureSensor, rTarget := _rCMAtTarget, eMode := E_CompareMode.GREATER_THAN, tTimeout := _tCMPressureTimeout, sNodeName := 'WaitCMAtTarget');
    _seq.AddChild(stepWaitCMAtTarget);

    // Engage PCV back-pressure control to the operating target before the HM pressure waits.
    stepSetPCVOperating.Init(ipController := _ipPressureController, rSetpoint := _rHMTarget, sNodeName := 'SetPCVOperating');
    _seq.AddChild(stepSetPCVOperating);

    stepWaitHMBelowTarget.Init(ipSensor := _ipHMPressureSensor, rTarget := _rHMTarget, eMode := E_CompareMode.LESS_THAN, tTimeout := _tHMPressureTimeout, sNodeName := 'WaitHMBelowTarget');
    _seq.AddChild(stepWaitHMBelowTarget);

    stepOpenCMBubbler.Init(ipValve := _ipCMBubblerValve, sNodeName := 'OpenCMBubbler');
    _seq.AddChild(stepOpenCMBubbler);

    stepWaitHMAtTarget.Init(ipSensor := _ipHMPressureSensor, rTarget := _rHMTarget, rTolerance := _rHMTolerance, eMode := E_CompareMode.WITHIN_TOLERANCE, tTimeout := _tHMPressureTimeout, sNodeName := 'WaitHMAtTarget');
    _seq.AddChild(stepWaitHMAtTarget);

    stepSetMFCTarget.Init(ipController := _ipMFCController, rSetpoint := _rFinalFlow, sNodeName := 'SetMFCTarget');
    _seq.AddChild(stepSetMFCTarget);
END_METHOD

PROPERTY PUBLIC NodeName : STRING(50)
    GET
        NodeName := _seq.sName;
    END_GET
    SET
        _seq.sName := NodeName;
    END_SET
END_PROPERTY

METHOD Tick : ST_NodeResult
    IF NOT _bInitialized THEN
        Tick.eStatus := E_NodeStatus.FAILURE;
        Tick.bHasError := TRUE;
        Tick.stError.eErrorId := E_ErrorId.ERR_GEN_INITIALIZATION;
        Tick.stError.sSource := 'FB_GasStartSequence';
        Tick.stError.sMessage := 'Init must be called before Tick';
        Tick.sDescription := Tick.stError.sMessage;
        RETURN;
    END_IF

    IF NOT _bParamsConfigured THEN
        Tick.eStatus := E_NodeStatus.FAILURE;
        Tick.bHasError := TRUE;
        Tick.stError.eErrorId := E_ErrorId.ERR_GEN_NOT_CONFIGURED;
        Tick.stError.sSource := 'FB_GasStartSequence';
        Tick.stError.sMessage := 'SetParams must be called before Tick';
        Tick.sDescription := Tick.stError.sMessage;
        RETURN;
    END_IF

    Tick := _seq.Tick();
END_METHOD

{attribute 'estimated-stack-usage' := '500'}
METHOD Reset : BOOL
    Reset := _seq.Reset();
END_METHOD

{attribute 'estimated-stack-usage' := '500'}
METHOD Halt
    _seq.Halt();
END_METHOD

END_FUNCTION_BLOCK

(* ---- FB_GasStopSequence.st ---- *)
(*
FB_GasStopSequence
Shuts down gas flow for one side. Parallel shutdown of manifold sections.
Bubbler array sized at compile-time upper bound (5); actual count comes
from provider.GetMaxBubblerCount() at runtime.
*)
FUNCTION_BLOCK FB_GasStopSequence IMPLEMENTS I_TreeNode
VAR
    _seq : FB_SequenceNode;
    // Delivery path shutdown
    stepCloseNozzleIso : FB_CloseValveNode;
    stepClosePCV       : FB_SetControllerNode;

    // HM shutdown (parallel)
    stepHMShutdown       : FB_ParallelNode;
    stepsCloseHMBubbler  : ARRAY[1..5] OF FB_CloseValveNode;
    stepCloseHMPurge     : FB_CloseValveNode;
    stepCloseHMVacuumIso : FB_CloseValveNode;

    // CM shutdown (parallel)
    stepCMShutdown       : FB_ParallelNode;
    stepsCloseCMBubbler  : ARRAY[1..5] OF FB_CloseValveNode;
    stepCloseCMPurge     : FB_CloseValveNode;
    stepCloseCMVacuumIso : FB_CloseValveNode;

    // Gas inlet shutdown (parallel)
    stepGasInletShutdown : FB_ParallelNode;
    stepsCloseGasIso     : ARRAY[1..5] OF FB_CloseValveNode;
    stepZeroMFC          : FB_SetControllerNode;

    // Internal state
    _bInitialized    : BOOL := FALSE;
    _eSide           : E_GasSide;
END_VAR

METHOD PUBLIC Init : BOOL
VAR_INPUT
    ipProvider : I_HardwareProvider;
    eSide      : E_GasSide;
END_VAR
VAR
    ipValve      : I_Valve;
    ipController : I_Controller;
    nMaxBubblers : DINT;
    i            : DINT;
END_VAR
    IF _bInitialized THEN
        IF _eSide = eSide THEN
            Init := TRUE;
            RETURN;
        END_IF
        _seq.ClearChildren();
        _bInitialized := FALSE;
    END_IF

    IF ipProvider = 0 THEN
        GVL_ErrorLogger.Logger.LogError('FB_GasStopSequence', E_ErrorId.ERR_GEN_NULL_POINTER, 'Provider is null');
        RETURN;
    END_IF

    nMaxBubblers := ipProvider.GetMaxBubblerCount(eSide);

    stepHMShutdown.ClearChildren();
    stepCMShutdown.ClearChildren();
    stepGasInletShutdown.ClearChildren();

    // Delivery path
    ipValve := ipProvider.GetNozzleIsoValve(eSide);
    stepCloseNozzleIso.Init(ipValve, sNodeName := 'CloseNozzleIso');
    _seq.AddChild(stepCloseNozzleIso);

    ipController := ipProvider.GetPressureController(eSide);
    stepClosePCV.Init(ipController := ipController, rSetpoint := GVL_SequenceConstants.PCV_CLOSED_SETPOINT, sNodeName := 'ClosePCV');
    _seq.AddChild(stepClosePCV);

    // HM shutdown
    ipValve := ipProvider.GetHMVacuumIsoValve(eSide);
    stepCloseHMVacuumIso.Init(ipValve, sNodeName := 'CloseHMVacIso');
    stepHMShutdown.AddChild(stepCloseHMVacuumIso);

    ipValve := ipProvider.GetHMPurgeValve(eSide);
    stepCloseHMPurge.Init(ipValve, sNodeName := 'CloseHMPurge');
    stepHMShutdown.AddChild(stepCloseHMPurge);

    FOR i := 1 TO nMaxBubblers DO
        ipValve := ipProvider.GetHMBubblerValve(eSide, i);
        IF ipValve <> 0 THEN
            stepsCloseHMBubbler[i].Init(ipValve);
            stepsCloseHMBubbler[i].sName := CONCAT('CloseHMBubbler_', TO_STRING(i));
            stepHMShutdown.AddChild(stepsCloseHMBubbler[i]);
        END_IF
    END_FOR

    stepHMShutdown.sName := 'HM_Shutdown';
    _seq.AddChild(stepHMShutdown);

    // CM shutdown
    ipValve := ipProvider.GetCMVacuumIsoValve(eSide);
    stepCloseCMVacuumIso.Init(ipValve, sNodeName := 'CloseCMVacIso');
    stepCMShutdown.AddChild(stepCloseCMVacuumIso);

    ipValve := ipProvider.GetCMPurgeValve(eSide);
    stepCloseCMPurge.Init(ipValve, sNodeName := 'CloseCMPurge');
    stepCMShutdown.AddChild(stepCloseCMPurge);

    FOR i := 1 TO nMaxBubblers DO
        ipValve := ipProvider.GetCMBubblerValve(eSide, i);
        IF ipValve <> 0 THEN
            stepsCloseCMBubbler[i].Init(ipValve);
            stepsCloseCMBubbler[i].sName := CONCAT('CloseCMBubbler_', TO_STRING(i));
            stepCMShutdown.AddChild(stepsCloseCMBubbler[i]);
        END_IF
    END_FOR

    stepCMShutdown.sName := 'CM_Shutdown';
    _seq.AddChild(stepCMShutdown);

    // Gas inlet shutdown
    ipController := ipProvider.GetMFCController(eSide);
    stepZeroMFC.Init(ipController := ipController, rSetpoint := 0.0, sNodeName := 'ZeroMFC');
    stepGasInletShutdown.AddChild(stepZeroMFC);

    FOR i := 1 TO nMaxBubblers DO
        ipValve := ipProvider.GetGasIsoValve(eSide, i);
        IF ipValve <> 0 THEN
            stepsCloseGasIso[i].Init(ipValve);
            stepsCloseGasIso[i].sName := CONCAT('CloseGasIso_', TO_STRING(i));
            stepGasInletShutdown.AddChild(stepsCloseGasIso[i]);
        END_IF
    END_FOR

    stepGasInletShutdown.sName := 'Inlet_Shutdown';
    _seq.AddChild(stepGasInletShutdown);

    _seq.sName := CONCAT('GasStop_', TO_STRING(eSide));
    _eSide := eSide;
    _bInitialized := TRUE;
    Init := TRUE;
END_METHOD

PROPERTY PUBLIC NodeName : STRING(50)
    GET
        NodeName := _seq.sName;
    END_GET
    SET
        _seq.sName := NodeName;
    END_SET
END_PROPERTY

METHOD Tick : ST_NodeResult
    IF NOT _bInitialized THEN
        Tick.eStatus := E_NodeStatus.FAILURE;
        Tick.bHasError := TRUE;
        Tick.stError.eErrorId := E_ErrorId.ERR_GEN_INITIALIZATION;
        Tick.stError.sSource := 'FB_GasStopSequence';
        Tick.stError.sMessage := 'Init must be called before Tick';
        Tick.sDescription := Tick.stError.sMessage;
        RETURN;
    END_IF

    Tick := _seq.Tick();
END_METHOD

{attribute 'estimated-stack-usage' := '500'}
METHOD Reset : BOOL
    Reset := _seq.Reset();
END_METHOD

{attribute 'estimated-stack-usage' := '500'}
METHOD Halt
    _seq.Halt();
END_METHOD

END_FUNCTION_BLOCK

(* ---- FB_HeatingSequence.st ---- *)
(*
FB_HeatingSequence
Sets up temperature gradient for gas delivery path: HM -> Umbilical -> Head.

One-shot: on first tick it enables the selected controllers and writes their
setpoints, then continuously reports SUCCESS while monitoring controller errors.

TEMPERATURE GRADIENT:
  HM (Combiner)     = combinerTemp (from payload)
  Umbilical (Start) = (combinerTemp + headTemp) / 2.0
  Head              = headTemp (from payload)

ENABLE MODES:
  0 = Both sides  1 = A-Only  2 = B-Only  3 = None
*)
FUNCTION_BLOCK FB_HeatingSequence IMPLEMENTS I_TreeNode
VAR
    // Internal State
    _bInitialized : BOOL := FALSE;
    _bApplied     : BOOL := FALSE;
    _bParamsConfigured : BOOL := FALSE;

    // Controller References
    _ipHM_A  : I_Controller;
    _ipHM_B  : I_Controller;
    _ipUmb_A : I_Controller;
    _ipUmb_B : I_Controller;
    _ipHead  : I_Controller;

    // Parameters (from SetParams)
    _rHMTemp_A   : LREAL;
    _rHMTemp_B   : LREAL;
    _rUmbTemp_A  : LREAL;
    _rUmbTemp_B  : LREAL;
    _rHeadTemp   : LREAL;
    _nEnableMode : INT;
    _bEnableA    : BOOL := FALSE;   // TRUE when A-side controllers are active (modes 0 or 1)
    _bEnableB    : BOOL := FALSE;   // TRUE when B-side controllers are active (modes 0 or 2)

    // Status
    _sErrorMsg : STRING(255);
END_VAR

METHOD PUBLIC Init : BOOL
VAR_INPUT
    ipProvider : I_HardwareProvider;
END_VAR
    _bInitialized := FALSE;
    _bApplied := FALSE;
    _bParamsConfigured := FALSE;
    _sErrorMsg := '';

    IF ipProvider = 0 THEN
        GVL_ErrorLogger.Logger.LogError('FB_HeatingSequence', E_ErrorId.ERR_GEN_NULL_POINTER, 'Provider is null');
        RETURN;
    END_IF

    _ipHM_A := ipProvider.GetHMTemperatureController(E_GasSide.A_SIDE);
    _ipHM_B := ipProvider.GetHMTemperatureController(E_GasSide.B_SIDE);
    _ipUmb_A := ipProvider.GetUmbilicalTemperatureController(E_GasSide.A_SIDE);
    _ipUmb_B := ipProvider.GetUmbilicalTemperatureController(E_GasSide.B_SIDE);
    _ipHead := ipProvider.GetHeadTemperatureController();

    IF _ipHead = 0 THEN
        GVL_ErrorLogger.Logger.LogError('FB_HeatingSequence', E_ErrorId.ERR_GEN_NULL_POINTER, 'Head controller not found');
        RETURN;
    END_IF

    _bInitialized := TRUE;
    Init := TRUE;
END_METHOD

METHOD PUBLIC SetParams
VAR_INPUT
    stCmd : ST_CmdSetTemperatureGradient;
END_VAR
    IF NOT _bInitialized THEN RETURN; END_IF

    _rHMTemp_A := REAL_TO_LREAL(stCmd.precursorCombiner);
    _rHMTemp_B := REAL_TO_LREAL(stCmd.reactantCombiner);
    _rHeadTemp := REAL_TO_LREAL(stCmd.headTemp);

    _rUmbTemp_A := (_rHMTemp_A + _rHeadTemp) / 2.0;
    _rUmbTemp_B := (_rHMTemp_B + _rHeadTemp) / 2.0;

    _nEnableMode := stCmd.enableMode;
    _bEnableA    := (stCmd.enableMode = 0 OR stCmd.enableMode = 1);
    _bEnableB    := (stCmd.enableMode = 0 OR stCmd.enableMode = 2);
    _bParamsConfigured := TRUE;
END_METHOD

METHOD PUBLIC Tick : ST_NodeResult
    IF NOT _bInitialized THEN
        Tick.eStatus := E_NodeStatus.FAILURE;
        Tick.bHasError := TRUE;
        Tick.stError.eErrorId := E_ErrorId.ERR_GEN_INITIALIZATION;
        Tick.stError.sSource := 'FB_HeatingSequence';
        Tick.stError.sMessage := 'Init must be called before Tick';
        Tick.sDescription := Tick.stError.sMessage;
        RETURN;
    END_IF

    IF NOT _bParamsConfigured THEN
        Tick.eStatus := E_NodeStatus.FAILURE;
        Tick.bHasError := TRUE;
        Tick.stError.eErrorId := E_ErrorId.ERR_GEN_NOT_CONFIGURED;
        Tick.stError.sSource := 'FB_HeatingSequence';
        Tick.stError.sMessage := 'SetParams must be called before Tick';
        Tick.sDescription := Tick.stError.sMessage;
        RETURN;
    END_IF

    // First tick: apply enable + setpoints once, then return RUNNING immediately.
    // DO NOT check _HeatingComplete() on the same tick we call Enable()/SetSetpoint().
    // FB_HeatZone.Execute() runs before the orchestrator in the PLC task; its cached
    // _stCtrlStatus still reflects _bEnabledCmd = FALSE from the previous scan.
    // Although _HeatingComplete() explicitly blocks while Head bEnabled=FALSE (so it
    // would not complete prematurely), returning RUNNING here gives Execute() at least
    // one scan cycle to process the Enable() command before the first completion check.
    IF NOT _bApplied THEN
        _EnableControllers(_bEnableA, _bEnableB);
        _SetSetpoints(_bEnableA, _bEnableB);
        _bApplied := TRUE;
        Tick.eStatus := E_NodeStatus.RUNNING;
        Tick.rProgress := 0.0;
        Tick.sDescription := 'Applying setpoints...';
        RETURN;
    END_IF

    // Error check runs every tick — controller faults after apply still fail the node.
    IF _CheckForErrors() THEN
        Tick.eStatus := E_NodeStatus.FAILURE;
        Tick.bHasError := TRUE;
        Tick.stError.eErrorId := E_ErrorId.ERR_GEN_INTERNAL;
        Tick.stError.sSource := 'FB_HeatingSequence';
        Tick.stError.sMessage := _sErrorMsg;
        Tick.sDescription := _sErrorMsg;
        RETURN;
    END_IF

    // Stay RUNNING until heating is physically complete: Head at setpoint (anchor)
    // and measured temperature gradient established for each active side.
    // sDescription carries live measured values so ramp progress is visible in telemetry.
    IF NOT _HeatingComplete() THEN
        Tick.eStatus := E_NodeStatus.RUNNING;
        Tick.rProgress := 0.0;
        Tick.sDescription := _BuildGradientStatus();
        RETURN;
    END_IF

    Tick.eStatus := E_NodeStatus.SUCCESS;
    Tick.rProgress := 100.0;
    Tick.sDescription := 'Heating Complete';
END_METHOD

METHOD PUBLIC Reset : BOOL
    _bApplied := FALSE;
    _sErrorMsg := '';

    _ResetIfErrored(_ipHM_A);
    _ResetIfErrored(_ipHM_B);
    _ResetIfErrored(_ipUmb_A);
    _ResetIfErrored(_ipUmb_B);
    _ResetIfErrored(_ipHead);

    Reset := TRUE;
END_METHOD

METHOD PUBLIC Halt
    Reset();
END_METHOD

PROPERTY PUBLIC NodeName : STRING(50)
    GET
        NodeName := 'HeatingSequence';
    END_GET
END_PROPERTY

METHOD PRIVATE _EnableControllers
VAR_INPUT
    bEnableA : BOOL;
    bEnableB : BOOL;
END_VAR
    IF _ipHM_A <> 0 THEN
        _ipHM_A.Enable(bEnableA);
    END_IF
    IF _ipUmb_A <> 0 THEN
        _ipUmb_A.Enable(bEnableA);
    END_IF
    IF _ipHM_B <> 0 THEN
        _ipHM_B.Enable(bEnableB);
    END_IF
    IF _ipUmb_B <> 0 THEN
        _ipUmb_B.Enable(bEnableB);
    END_IF
    IF _ipHead <> 0 THEN
        _ipHead.Enable(bEnableA OR bEnableB);
    END_IF
END_METHOD

METHOD PRIVATE _SetSetpoints
VAR_INPUT
    bEnableA : BOOL;
    bEnableB : BOOL;
END_VAR
    IF bEnableA THEN
        IF _ipHM_A <> 0 THEN
            _ipHM_A.SetSetpoint(_rHMTemp_A);
        END_IF
        IF _ipUmb_A <> 0 THEN
            _ipUmb_A.SetSetpoint(_rUmbTemp_A);
        END_IF
    END_IF

    IF bEnableB THEN
        IF _ipHM_B <> 0 THEN
            _ipHM_B.SetSetpoint(_rHMTemp_B);
        END_IF
        IF _ipUmb_B <> 0 THEN
            _ipUmb_B.SetSetpoint(_rUmbTemp_B);
        END_IF
    END_IF

    IF _ipHead <> 0 AND (bEnableA OR bEnableB) THEN
        _ipHead.SetSetpoint(_rHeadTemp);
    END_IF
END_METHOD

METHOD PRIVATE _CheckForErrors : BOOL
    _sErrorMsg := '';
    IF _ControllerInError(_ipHM_A, 'HM A-Side') THEN _CheckForErrors := TRUE; RETURN; END_IF
    IF _ControllerInError(_ipUmb_A, 'Umbilical A-Side') THEN _CheckForErrors := TRUE; RETURN; END_IF
    IF _ControllerInError(_ipHM_B, 'HM B-Side') THEN _CheckForErrors := TRUE; RETURN; END_IF
    IF _ControllerInError(_ipUmb_B, 'Umbilical B-Side') THEN _CheckForErrors := TRUE; RETURN; END_IF
    IF _ControllerInError(_ipHead, 'Head') THEN _CheckForErrors := TRUE; RETURN; END_IF
    _CheckForErrors := FALSE;
END_METHOD

// Heating is physically complete when both conditions hold:
//   1. Head has reached its target setpoint — the high-temperature anchor of the gradient.
//      Until Head is enabled and at setpoint, checking the downstream gradient is premature.
//   2. The measured temperature ordering is correct for every active side:
//      Head.measured > Umbilical.measured > HM.measured
//
// HM and Umbilical are NOT required to reach their individual programmed setpoints.
// The gradient being established is the physical completion criterion — a zone that is
// colder than the one upstream of it would cause gas condensation in the delivery line.
METHOD PRIVATE _HeatingComplete : BOOL
VAR
    stHead : ST_ControllerStatus;
END_VAR
    // Mode 3 (ENABLE_NONE): no heating active, nothing to wait for.
    IF NOT _bEnableA AND NOT _bEnableB THEN
        _HeatingComplete := TRUE;
        RETURN;
    END_IF

    // Head must be enabled and at setpoint before declaring the gradient valid.
    stHead := _ipHead.GetStatus();
    IF NOT stHead.bEnabled OR NOT stHead.bAtSetpoint THEN
        RETURN;   // FALSE by default
    END_IF

    // Check the gradient for each active side.
    IF _bEnableA AND NOT _SideGradientCorrect(_ipHead, _ipUmb_A, _ipHM_A) THEN
        RETURN;
    END_IF
    IF _bEnableB AND NOT _SideGradientCorrect(_ipHead, _ipUmb_B, _ipHM_B) THEN
        RETURN;
    END_IF

    _HeatingComplete := TRUE;
END_METHOD

// Builds a human-readable snapshot of measured temperatures for every active side.
// Called from Tick() as sDescription while waiting, so live temperatures are visible
// in telemetry and the watch window without needing a separate diagnostic variable.
METHOD PRIVATE _BuildGradientStatus : STRING(255)
VAR
    sResult : STRING(255);
    stHead  : ST_ControllerStatus;
    stUmbA  : ST_ControllerStatus;
    stHMA   : ST_ControllerStatus;
    stUmbB  : ST_ControllerStatus;
    stHMB   : ST_ControllerStatus;
END_VAR
    stHead  := _ipHead.GetStatus();
    sResult := CONCAT('Gradient: Head=', LREAL_TO_STRING(stHead.rMeasuredValue));

    IF _bEnableA THEN
        stUmbA  := _ipUmb_A.GetStatus();
        stHMA   := _ipHM_A.GetStatus();
        sResult := CONCAT(sResult, CONCAT(' UmbA=', LREAL_TO_STRING(stUmbA.rMeasuredValue)));
        sResult := CONCAT(sResult, CONCAT(' HMA=',  LREAL_TO_STRING(stHMA.rMeasuredValue)));
    END_IF

    IF _bEnableB THEN
        stUmbB  := _ipUmb_B.GetStatus();
        stHMB   := _ipHM_B.GetStatus();
        sResult := CONCAT(sResult, CONCAT(' UmbB=', LREAL_TO_STRING(stUmbB.rMeasuredValue)));
        sResult := CONCAT(sResult, CONCAT(' HMB=',  LREAL_TO_STRING(stHMB.rMeasuredValue)));
    END_IF

    _BuildGradientStatus := sResult;
END_METHOD

// Checks that the measured temperature ordering along one gas-delivery side is correct:
//   Head > Umbilical > HM (Hot Manifold)
// This ordering ensures no zone is colder than the one upstream of it — a colder
// downstream zone would cause gas condensation inside the line.
// Uses rMeasuredValue (live sensor reading) rather than bAtSetpoint, because the
// gradient being established is the physical completion criterion, not whether each
// zone has individually converged to its programmed number.
METHOD PRIVATE _SideGradientCorrect : BOOL
VAR_INPUT
    ipHead : I_Controller;   // Head — highest temperature in the path
    ipUmb  : I_Controller;   // Umbilical — midpoint
    ipHM   : I_Controller;   // Hot Manifold — lowest temperature in the path
END_VAR
VAR
    stHead : ST_ControllerStatus;
    stUmb  : ST_ControllerStatus;
    stHM   : ST_ControllerStatus;
END_VAR
    IF ipHead = 0 OR ipUmb = 0 OR ipHM = 0 THEN
        RETURN;   // Any null pointer means gradient cannot be verified — block completion
    END_IF

    stHead := ipHead.GetStatus();
    stUmb  := ipUmb.GetStatus();
    stHM   := ipHM.GetStatus();

    // Strict greater-than matches the reference implementation.
    // Gradient holds when each zone is measurably warmer than the one behind it.
    _SideGradientCorrect := (stHead.rMeasuredValue > stUmb.rMeasuredValue)
                        AND (stUmb.rMeasuredValue  > stHM.rMeasuredValue);
END_METHOD

METHOD PRIVATE _ControllerInError : BOOL
VAR_INPUT
    ipCtrl : I_Controller;
    sLabel : STRING(80);
END_VAR
VAR
    stStatus : ST_ControllerStatus;
END_VAR
    IF ipCtrl = 0 THEN RETURN; END_IF
    stStatus := ipCtrl.GetStatus();
    IF stStatus.stError.eErrorId <> E_ErrorId.NO_ERROR THEN
        _sErrorMsg := CONCAT(sLabel, ' error');
        _ControllerInError := TRUE;
    END_IF
END_METHOD

METHOD PRIVATE _ResetIfErrored
VAR_INPUT
    ipCtrl : I_Controller;
END_VAR
VAR
    stStatus : ST_ControllerStatus;
END_VAR
    IF ipCtrl = 0 THEN RETURN; END_IF
    stStatus := ipCtrl.GetStatus();
    IF stStatus.stError.eErrorId <> E_ErrorId.NO_ERROR THEN
        ipCtrl.Reset();
    END_IF
END_METHOD

END_FUNCTION_BLOCK

(* ---- FB_MaintenancePurgeSequence.st ---- *)
(*
FB_MaintenancePurgeSequence
Complete maintenance purge for a specific bubbler (CM + HM + Umbilical regions).
Use when replacing bubblers or performing maintenance requiring full gas path purge.
*)
FUNCTION_BLOCK FB_MaintenancePurgeSequence IMPLEMENTS I_TreeNode
VAR
    _seq : FB_SequenceNode;
    // Steps
    stepPrepareExhaust : FB_PrepareExhaustSequence;
    stepBubblerPurgeCM : FB_BubblerPurgeCMSequence;
    stepDelayCMtoHM    : FB_WaitNode;
    stepBubblerPurgeHM : FB_BubblerPurgeHMSequence;
    stepDelayHMtoUmb   : FB_WaitNode;
    stepUmbilicalPurge : FB_MaintenancePurgeUmbilicalSequence;

    // Internal state
    _bInitialized    : BOOL := FALSE;
    _eSide           : E_GasSide;
    _nBubblerIndex   : DINT;
END_VAR

VAR CONSTANT
    PHASE_TRANSITION_DELAY : TIME := T#5S;
END_VAR

METHOD PUBLIC Init : BOOL
VAR_INPUT
    ipProvider    : I_HardwareProvider;
    eSide         : E_GasSide;
    nBubblerIndex : DINT;
END_VAR
    IF _bInitialized THEN
        IF _eSide = eSide AND _nBubblerIndex = nBubblerIndex THEN
            Init := TRUE;
            RETURN;
        END_IF
        _seq.ClearChildren();
        _bInitialized := FALSE;
    END_IF

    IF ipProvider = 0 THEN
        GVL_ErrorLogger.Logger.LogError('FB_MaintenancePurgeSequence', E_ErrorId.ERR_GEN_NULL_POINTER, 'Provider is null');
        RETURN;
    END_IF
    _eSide := eSide;
    _nBubblerIndex := nBubblerIndex;

    stepPrepareExhaust.Init(ipProvider, eSide);
    stepPrepareExhaust.NodeName := 'PrepareExhaust';
    _seq.AddChild(stepPrepareExhaust);

    stepBubblerPurgeCM.Init(ipProvider, eSide, nBubblerIndex);
    stepBubblerPurgeCM.NodeName := 'BubblerPurgeCM';
    _seq.AddChild(stepBubblerPurgeCM);

    stepDelayCMtoHM.Init(tWaitTime := PHASE_TRANSITION_DELAY, sNodeName := 'DelayCMtoHM');
    _seq.AddChild(stepDelayCMtoHM);

    stepBubblerPurgeHM.Init(ipProvider, eSide, nBubblerIndex);
    stepBubblerPurgeHM.NodeName := 'BubblerPurgeHM';
    _seq.AddChild(stepBubblerPurgeHM);

    stepDelayHMtoUmb.Init(tWaitTime := PHASE_TRANSITION_DELAY, sNodeName := 'DelayHMtoUmb');
    _seq.AddChild(stepDelayHMtoUmb);

    stepUmbilicalPurge.Init(ipProvider, eSide);
    stepUmbilicalPurge.NodeName := 'UmbilicalPurge';
    _seq.AddChild(stepUmbilicalPurge);

    _seq.sName := CONCAT(CONCAT('MaintenancePurge_Side', TO_STRING(eSide)), CONCAT('_Idx', TO_STRING(nBubblerIndex)));

    _bInitialized := TRUE;
    Init := TRUE;
END_METHOD

METHOD PUBLIC SetParams
VAR_INPUT
    stCmd : ST_CmdPurge;
END_VAR
    IF NOT _bInitialized THEN RETURN; END_IF

    // Phase 1: CM Purge parameters
    stepBubblerPurgeCM.SetParams(
        nPurgeCycles           := stCmd.coldManifoldPurgeCycles,
        rPurgeFlowRate         := REAL_TO_LREAL(stCmd.purgeGasFlow),
        rPurgePressure         := REAL_TO_LREAL(stCmd.purgeHighPressureLimit),
        rEvacuationPressure    := REAL_TO_LREAL(stCmd.purgeLowPressureLimit),
        tPressurizationTimeout := DINT_TO_TIME(stCmd.highPressureTimeout),
        tEvacuationTimeout     := DINT_TO_TIME(stCmd.lowPressureTimeout)
    );

    // Phase 3: HM Purge parameters (Final state = operating pressure)
    stepBubblerPurgeHM.SetParams(
        nPurgeCycles           := stCmd.hotManifoldPurgeCycles,
        rPurgeFlowRate         := REAL_TO_LREAL(stCmd.purgeGasFlow),
        rPurgePressure         := REAL_TO_LREAL(stCmd.purgeHighPressureLimit),
        rFinalPressure         := REAL_TO_LREAL(stCmd.hotManifoldOperatingPressure),
        rEvacuationPressure    := REAL_TO_LREAL(stCmd.purgeLowPressureLimit),
        tPressurizationTimeout := DINT_TO_TIME(stCmd.highPressureTimeout),
        tEvacuationTimeout     := DINT_TO_TIME(stCmd.lowPressureTimeout)
    );

    stepUmbilicalPurge.SetParams(
        rPurgeFlowRate      := REAL_TO_LREAL(stCmd.purgeGasFlow),
        rCMPressureTarget   := REAL_TO_LREAL(stCmd.purgeHighPressureLimit),
        rHMPressureTarget   := REAL_TO_LREAL(stCmd.purgeHighPressureLimit),
        rPCVSetpoint        := REAL_TO_LREAL(stCmd.hotManifoldOperatingPressure),
        tCMPressureTimeout  := DINT_TO_TIME(stCmd.highPressureTimeout),
        tHMPressureTimeout  := DINT_TO_TIME(stCmd.highPressureTimeout),
        tStabilizationDelay := DINT_TO_TIME(stCmd.stabilisationDelay),
        tPurgeDuration      := DINT_TO_TIME(stCmd.umbilicalFlushTime)
    );
END_METHOD

PROPERTY PUBLIC NodeName : STRING(50)
    GET
        NodeName := _seq.sName;
    END_GET
    SET
        _seq.sName := NodeName;
    END_SET
END_PROPERTY

METHOD Tick : ST_NodeResult
    IF NOT _bInitialized THEN
        Tick.eStatus := E_NodeStatus.FAILURE;
        Tick.bHasError := TRUE;
        Tick.stError.eErrorId := E_ErrorId.ERR_GEN_INITIALIZATION;
        Tick.stError.sSource := 'FB_MaintenancePurgeSequence';
        Tick.stError.sMessage := 'Init must be called before Tick';
        Tick.sDescription := Tick.stError.sMessage;
        RETURN;
    END_IF

    Tick := _seq.Tick();
END_METHOD

{attribute 'estimated-stack-usage' := '500'}
METHOD Reset : BOOL
    Reset := _seq.Reset();
END_METHOD

{attribute 'estimated-stack-usage' := '500'}
METHOD Halt
    _seq.Halt();
END_METHOD

END_FUNCTION_BLOCK

(* ---- FB_MaterialPurgeSequence.st ---- *)
(*
FB_MaterialPurgeSequence
Full material purge: Prepare exhaust -> HM purge cycles -> Umbilical purge -> Cleanup.
*)
FUNCTION_BLOCK FB_MaterialPurgeSequence IMPLEMENTS I_TreeNode
VAR
    _seq : FB_SequenceNode;
    // Phase 1: Prepare exhaust
    stepPrepareExhaust : FB_PrepareExhaustSequence;

    // Phase 2: HM purge (vacuum/pressurize cycles)
    stepHMPurge : FB_MaterialPurgeHMSequence;

    // Phase 3: Umbilical purge (push-to-atmosphere)
    stepUmbilicalPurge : FB_MaterialPurgeUmbilicalSequence;

    // Phase 4: Cleanup
    stepCleanup          : FB_ParallelNode;
    stepCloseHMPurge     : FB_CloseValveNode;
    stepCloseCMPurge     : FB_CloseValveNode;
    stepCloseExhaustPump : FB_CloseValveNode;
    stepZeroMFCFinal     : FB_SetControllerNode;

    // Internal state
    _bInitialized    : BOOL := FALSE;
    _eSide           : E_GasSide;
END_VAR

METHOD PUBLIC Init : BOOL
VAR_INPUT
    ipProvider : I_HardwareProvider;
    eSide      : E_GasSide;
END_VAR
VAR
    ipExhaustVacuumIso : I_Valve;
    ipHMPurge          : I_Valve;
    ipCMPurge          : I_Valve;
    ipMFC              : I_Controller;
END_VAR
    IF _bInitialized THEN
        IF _eSide = eSide THEN
            Init := TRUE;
            RETURN;
        END_IF
        _seq.ClearChildren();
        _bInitialized := FALSE;
    END_IF

    IF ipProvider = 0 THEN
        GVL_ErrorLogger.Logger.LogError('FB_MaterialPurgeSequence', E_ErrorId.ERR_GEN_NULL_POINTER, 'Provider is null');
        RETURN;
    END_IF
    _eSide := eSide;

    stepPrepareExhaust.Init(ipProvider := ipProvider, eSide := eSide);
    stepPrepareExhaust.NodeName := 'PrepareExhaust';
    _seq.AddChild(stepPrepareExhaust);

    stepHMPurge.Init(ipProvider := ipProvider, eSide := eSide);
    stepHMPurge.NodeName := 'HMPurge';
    _seq.AddChild(stepHMPurge);

    stepUmbilicalPurge.Init(ipProvider := ipProvider, eSide := eSide);
    stepUmbilicalPurge.NodeName := 'UmbilicalPurge';
    _seq.AddChild(stepUmbilicalPurge);

    // Cleanup phase
    stepCleanup.ClearChildren();

    ipHMPurge := ipProvider.GetHMPurgeValve(eSide);
    ipCMPurge := ipProvider.GetCMPurgeValve(eSide);
    ipExhaustVacuumIso := ipProvider.GetExhaustVacuumIsoValve();
    ipMFC := ipProvider.GetMFCController(eSide);

    stepCloseHMPurge.Init(ipHMPurge, sNodeName := 'CloseHMPurge');
    stepCleanup.AddChild(stepCloseHMPurge);

    stepCloseCMPurge.Init(ipCMPurge, sNodeName := 'CloseCMPurge');
    stepCleanup.AddChild(stepCloseCMPurge);

    stepCloseExhaustPump.Init(ipExhaustVacuumIso, sNodeName := 'CloseExhaustPump');
    stepCleanup.AddChild(stepCloseExhaustPump);

    stepZeroMFCFinal.Init(ipController := ipMFC, rSetpoint := 0.0, sNodeName := 'ZeroMFC');
    stepCleanup.AddChild(stepZeroMFCFinal);

    stepCleanup.sName := 'Cleanup';
    _seq.AddChild(stepCleanup);

    _seq.sName := CONCAT('MaterialPurge_', TO_STRING(eSide));
    _bInitialized := TRUE;
    Init := TRUE;
END_METHOD

METHOD PUBLIC SetParams
VAR_INPUT
    stCmd : ST_CmdPurge;
END_VAR
    IF NOT _bInitialized THEN RETURN; END_IF

    stepHMPurge.SetParams(
        nPurgeCycles           := stCmd.hotManifoldPurgeCycles,
        rPurgeFlowRate         := REAL_TO_LREAL(stCmd.purgeGasFlow),
        rPurgePressure         := REAL_TO_LREAL(stCmd.purgeHighPressureLimit),
        rFinalPressure         := REAL_TO_LREAL(stCmd.hotManifoldOperatingPressure),
        rEvacuationPressure    := REAL_TO_LREAL(stCmd.purgeLowPressureLimit),
        tPressurizationTimeout := DINT_TO_TIME(stCmd.highPressureTimeout),
        tEvacuationTimeout     := DINT_TO_TIME(stCmd.lowPressureTimeout)
    );

    stepUmbilicalPurge.SetParams(
        rPurgeFlowRate      := REAL_TO_LREAL(stCmd.purgeGasFlow),
        rCMPressureTarget   := REAL_TO_LREAL(stCmd.purgeHighPressureLimit),
        rHMPressureTarget   := REAL_TO_LREAL(stCmd.purgeHighPressureLimit),
        rPCVSetpoint        := REAL_TO_LREAL(stCmd.hotManifoldOperatingPressure),
        tCMPressureTimeout  := DINT_TO_TIME(stCmd.highPressureTimeout),
        tHMPressureTimeout  := DINT_TO_TIME(stCmd.highPressureTimeout),
        tStabilizationDelay := DINT_TO_TIME(stCmd.stabilisationDelay),
        tPurgeDuration      := DINT_TO_TIME(stCmd.umbilicalFlushTime)
    );
END_METHOD

PROPERTY PUBLIC NodeName : STRING(50)
    GET
        NodeName := _seq.sName;
    END_GET
    SET
        _seq.sName := NodeName;
    END_SET
END_PROPERTY

METHOD Tick : ST_NodeResult
    IF NOT _bInitialized THEN
        Tick.eStatus := E_NodeStatus.FAILURE;
        Tick.bHasError := TRUE;
        Tick.stError.eErrorId := E_ErrorId.ERR_GEN_INITIALIZATION;
        Tick.stError.sSource := 'FB_MaterialPurgeSequence';
        Tick.stError.sMessage := 'Init must be called before Tick';
        Tick.sDescription := Tick.stError.sMessage;
        RETURN;
    END_IF

    Tick := _seq.Tick();
END_METHOD

{attribute 'estimated-stack-usage' := '500'}
METHOD Reset : BOOL
    Reset := _seq.Reset();
END_METHOD

{attribute 'estimated-stack-usage' := '500'}
METHOD Halt
    _seq.Halt();
END_METHOD

END_FUNCTION_BLOCK

(* ---- FB_SequenceOrchestrator.st ---- *)
(*
FB_SequenceOrchestrator — Shared sequence dispatch and execution engine.

All sequence FBs, types, and enums used here live in Lib, so this FB has
no App-level dependencies and compiles independently of any machine target.

USAGE (thin PROGRAM wrapper pattern):
  PROGRAM PRG_Sequence
  VAR
      fbOrchestrator : FB_SequenceOrchestrator;
  END_VAR
      fbOrchestrator();
  // Delegate methods call fbOrchestrator.XxxMethod()

ADDING A NEW SEQUENCE:
  1. Create FB_MySequence IMPLEMENTS I_TreeNode in Lib/Sequences/
  2. Add instance to VAR: _fbMySeq : FB_MySequence
  3. Add public dispatch method that calls _fbMySeq.Init() + _Start()
  4. Add the E_Sequence enum value to Lib/Sequences/Types/E_Sequence.st
*)
FUNCTION_BLOCK FB_SequenceOrchestrator
VAR
    eActiveSequence     : E_Sequence := E_Sequence.None;
    sStatus             : STRING(255) := 'Ready';
    bBusy               : BOOL;
    bDone               : BOOL;
    bError              : BOOL;
    rProgress           : REAL := 0.0;
    stLastError         : ST_Error;
    nLastPurgedBubblerA : INT := 0;     // Last bubbler index purged on A-side (precursor)
    nLastPurgedBubblerB : INT := 0;     // Last bubbler index purged on B-side (reactant)
END_VAR
VAR
    _ipProvider       : I_HardwareProvider;
    _bConfigured      : BOOL := FALSE;
    _ipActiveSequence : I_TreeNode;
    _stLastResult     : ST_NodeResult;
    _eSide            : E_GasSide;
    _nBubblerIndex    : DINT;

    // Shared sequences
    _fbGasStart         : FB_GasStartSequence;
    _fbGasStop          : FB_GasStopSequence;
    _fbSystemStop       : FB_SystemStopSequence;
    _fbMaterialPurge    : FB_MaterialPurgeSequence;
    _fbBubblerPurge     : FB_BubblerPurgeSequence;
    _fbMaintenancePurge : FB_MaintenancePurgeSequence;
    _fbHeating          : FB_HeatingSequence;
    _fbChuckHold        : FB_ChuckVacuumHoldSequence;
    _fbChuckRelease     : FB_ChuckVacuumReleaseSequence;

    // Extended sequences (types and FBs are in Lib; not all machines use them)
    _fbSpotDeposition   : FB_SpotDepositionSequence;
    _fbBubblerLeakTest  : FB_BubblerLeakTestSequence;
END_VAR

    IF NOT _bConfigured THEN
        sStatus := 'Not configured';
        RETURN;
    END_IF

    IF eActiveSequence <> E_Sequence.None AND eActiveSequence <> E_Sequence.Error THEN
        _ExecuteSequence();
    END_IF

END_FUNCTION_BLOCK

// =============================================================================
// PUBLIC API
// =============================================================================

METHOD PUBLIC Configure : BOOL
VAR_INPUT
    ipProvider : I_HardwareProvider;
END_VAR
    IF ipProvider = 0 THEN RETURN; END_IF
    _ipProvider  := ipProvider;
    _bConfigured := TRUE;
    sStatus      := 'Ready';
    Configure    := TRUE;
END_METHOD

METHOD PUBLIC GetStatus : ST_SequenceStatus
    GetStatus.eActiveSequence     := eActiveSequence;
    GetStatus.bBusy               := bBusy;
    GetStatus.bDone               := bDone;
    GetStatus.bError              := bError;
    GetStatus.sStatusMessage      := sStatus;
    GetStatus.rProgress           := rProgress;
    GetStatus.stLastError         := stLastError;
    GetStatus.nLastPurgedBubblerA := nLastPurgedBubblerA;
    GetStatus.nLastPurgedBubblerB := nLastPurgedBubblerB;
END_METHOD

METHOD PUBLIC ErrorAcknowledge : BOOL
    IF eActiveSequence <> E_Sequence.Error THEN RETURN; END_IF
    _ResetState();
    ErrorAcknowledge := TRUE;
END_METHOD

METHOD PUBLIC AcknowledgeDone : BOOL
    // Clears the latched bDone once a successful completion has been observed.
    IF NOT bDone THEN RETURN; END_IF
    bDone           := FALSE;
    sStatus         := 'Ready';
    AcknowledgeDone := TRUE;
END_METHOD

METHOD PUBLIC StartBubblerFlow : BOOL
VAR_INPUT
    stParams : ST_CmdStartBubblerFlow;
END_VAR
VAR
    eSide : E_GasSide;
    eSeq  : E_Sequence;
END_VAR
    IF NOT _CanStart() THEN RETURN; END_IF
    IF NOT _MapSide(nSide := stParams.side, eSide => eSide) THEN RETURN; END_IF

    eSeq := SEL(eSide = E_GasSide.A_SIDE, E_Sequence.ReactantStart, E_Sequence.PrecursorStart);

    IF NOT _fbGasStart.Init(ipProvider := _ipProvider, eSide := eSide, nBubblerIndex := stParams.bubblerIndex) THEN
        _SetError('GasStart init failed');
        RETURN;
    END_IF
    _fbGasStart.SetParams(stParams);
    _ipActiveSequence := _fbGasStart;
    _eSide            := eSide;
    _nBubblerIndex    := stParams.bubblerIndex;
    _Start(eSeq, 'Starting bubbler flow...');
    StartBubblerFlow := TRUE;
END_METHOD

METHOD PUBLIC StopBubblerFlow : BOOL
VAR_INPUT
    stParams : ST_CmdStopBubblerFlow;
END_VAR
VAR
    eSide : E_GasSide;
    eSeq  : E_Sequence;
END_VAR
    IF NOT _CanStart() THEN RETURN; END_IF
    IF NOT _MapSide(nSide := stParams.side, eSide => eSide) THEN RETURN; END_IF

    eSeq := SEL(eSide = E_GasSide.A_SIDE, E_Sequence.ReactantStop, E_Sequence.PrecursorStop);

    IF NOT _fbGasStop.Init(ipProvider := _ipProvider, eSide := eSide) THEN
        _SetError('GasStop init failed');
        RETURN;
    END_IF
    _ipActiveSequence := _fbGasStop;
    _eSide            := eSide;
    _Start(eSeq, 'Stopping bubbler flow...');
    StopBubblerFlow := TRUE;
END_METHOD

METHOD PUBLIC SystemStop : BOOL
    SystemStop := _InitiateSystemStop('System stop');
END_METHOD

METHOD PUBLIC EmergencyStop : BOOL
    // Immediate safe-state halt. Unlike SystemStop, this does NOT run the
    // multi-step FB_SystemStopSequence; it halts the active sequence right away
    // (Halt cascades hardware to its safe state) and returns to IDLE.
    _AbortCurrentSequence();
    _ResetState();
    sStatus       := 'Emergency stop';
    EmergencyStop := TRUE;
END_METHOD

METHOD PUBLIC StartPurge : BOOL
VAR_INPUT
    stParams : ST_CmdPurge;
END_VAR
VAR
    eSide : E_GasSide;
    eSeq  : E_Sequence;
END_VAR
    IF NOT _CanStart() THEN RETURN; END_IF
    IF NOT _MapSide(nSide := stParams.side, eSide => eSide) THEN RETURN; END_IF

    eSeq           := SEL(eSide = E_GasSide.A_SIDE, E_Sequence.PurgeReactant, E_Sequence.PurgePrecursor);
    _nBubblerIndex := INT_TO_DINT(stParams.bubbler);
    _eSide         := eSide;

    CASE stParams.mode OF
        E_PurgeMode.ChangeMaterial:
            IF NOT _fbMaterialPurge.Init(ipProvider := _ipProvider, eSide := eSide) THEN
                _SetError('MaterialPurge init failed');
                RETURN;
            END_IF
            _fbMaterialPurge.SetParams(stParams);
            _ipActiveSequence := _fbMaterialPurge;
            _Start(eSeq, 'Material purge...');

        E_PurgeMode.ReplaceBubbler:
            IF NOT _fbBubblerPurge.Init(ipProvider := _ipProvider, eSide := eSide, nBubblerIndex := INT_TO_DINT(stParams.bubbler)) THEN
                _SetError('BubblerPurge init failed');
                RETURN;
            END_IF
            _fbBubblerPurge.SetParams(stParams);
            _ipActiveSequence := _fbBubblerPurge;
            _Start(eSeq, 'Bubbler purge...');

        E_PurgeMode.Maintenance:
            IF NOT _fbMaintenancePurge.Init(ipProvider := _ipProvider, eSide := eSide, nBubblerIndex := INT_TO_DINT(stParams.bubbler)) THEN
                _SetError('MaintenancePurge init failed');
                RETURN;
            END_IF
            _fbMaintenancePurge.SetParams(stParams);
            _ipActiveSequence := _fbMaintenancePurge;
            _Start(eSeq, 'Maintenance purge...');
    ELSE
        sStatus := 'Invalid purge mode';
        RETURN;
    END_CASE
    StartPurge := TRUE;
END_METHOD

METHOD PUBLIC StartHeating : BOOL
VAR_INPUT
    stParams : ST_CmdSetTemperatureGradient;
END_VAR
    IF NOT _CanStart() THEN RETURN; END_IF

    IF NOT _fbHeating.Init(ipProvider := _ipProvider) THEN
        _SetError('Heating init failed');
        RETURN;
    END_IF
    _fbHeating.SetParams(stParams);
    _ipActiveSequence := _fbHeating;
    _Start(E_Sequence.HeatingStart, 'Setting temperature gradient...');
    StartHeating := TRUE;
END_METHOD

METHOD PUBLIC StartChuckVacuumHold : BOOL
VAR_INPUT
    stParams : ST_ChuckVacuumHold;
END_VAR
    IF NOT _CanStart() THEN RETURN; END_IF

    IF NOT _fbChuckHold.Init(ipProvider := _ipProvider) THEN
        _SetError('ChuckVacuumHold init failed');
        RETURN;
    END_IF
    _fbChuckHold.SetParams(stParams);
    _ipActiveSequence := _fbChuckHold;
    _Start(E_Sequence.ChuckVacuumHold, 'Applying chuck vacuum...');
    StartChuckVacuumHold := TRUE;
END_METHOD

METHOD PUBLIC StartChuckVacuumRelease : BOOL
VAR_INPUT
    stParams : ST_ChuckVacuumRelease;
END_VAR
    IF NOT _CanStart() THEN RETURN; END_IF

    IF NOT _fbChuckRelease.Init(ipProvider := _ipProvider) THEN
        _SetError('ChuckVacuumRelease init failed');
        RETURN;
    END_IF
    _fbChuckRelease.SetParams(stParams);
    _ipActiveSequence := _fbChuckRelease;
    _Start(E_Sequence.ChuckVacuumRelease, 'Releasing chuck vacuum...');
    StartChuckVacuumRelease := TRUE;
END_METHOD

METHOD PUBLIC StartSpotDeposition : BOOL
VAR_INPUT
    stParams : ST_CmdSpotDeposition;
END_VAR
    IF NOT _CanStart() THEN RETURN; END_IF

    IF NOT _fbSpotDeposition.Init(ipProvider := _ipProvider) THEN
        _SetError('SpotDeposition init failed');
        RETURN;
    END_IF
    _fbSpotDeposition.SetParams(stParams);
    _ipActiveSequence := _fbSpotDeposition;
    _Start(E_Sequence.SpotDeposition, 'Spot deposition...');
    StartSpotDeposition := TRUE;
END_METHOD

METHOD PUBLIC StartBubblerLeakTest : BOOL
VAR_INPUT
    stParams : ST_CmdBubblerLeakTest;
END_VAR
VAR
    eSide : E_GasSide;
END_VAR
    IF NOT _CanStart() THEN RETURN; END_IF
    IF NOT _MapSide(nSide := stParams.side, eSide => eSide) THEN RETURN; END_IF

    IF NOT _fbBubblerLeakTest.Init(ipProvider := _ipProvider, eSide := eSide, nBubblerIndex := stParams.bubblerIndex) THEN
        _SetError('BubblerLeakTest init failed');
        RETURN;
    END_IF
    _fbBubblerLeakTest.SetParams(stParams);
    _ipActiveSequence := _fbBubblerLeakTest;
    _eSide            := eSide;
    _nBubblerIndex    := stParams.bubblerIndex;
    _Start(E_Sequence.BubblerLeakTest, 'Bubbler leak test...');
    StartBubblerLeakTest := TRUE;
END_METHOD

// =============================================================================
// PRIVATE — Execution Engine
// =============================================================================

METHOD PRIVATE _CanStart : BOOL
    CASE eActiveSequence OF
        E_Sequence.None:
            _CanStart := TRUE;
        E_Sequence.Error:
            sStatus := 'Error not acknowledged';
    ELSE
        sStatus := 'Sequence already running';
    END_CASE
END_METHOD

METHOD PRIVATE _Start
VAR_INPUT
    eSeq : E_Sequence;
    sMsg : STRING(255);
END_VAR
    _ipActiveSequence.Reset();
    eActiveSequence := eSeq;
    bBusy           := TRUE;
    bDone           := FALSE;
    bError          := FALSE;
    rProgress       := 0.0;
    sStatus         := sMsg;
END_METHOD

METHOD PRIVATE _ExecuteSequence
    IF _ipActiveSequence = 0 THEN
        _SetError('No active sequence', E_ErrorId.ERR_GEN_NULL_POINTER);
        RETURN;
    END_IF

    _stLastResult := _ipActiveSequence.Tick();
    sStatus       := _stLastResult.sDescription;

    CASE _stLastResult.eStatus OF
        E_NodeStatus.RUNNING:
            bBusy     := TRUE;
            rProgress := _stLastResult.rProgress;
            IF sStatus = '' THEN sStatus := 'Running...'; END_IF

        E_NodeStatus.SUCCESS:
            _UpdateLastPurgedBubbler();
            _CompleteSequence();

        E_NodeStatus.FAILURE:
            IF sStatus = '' THEN sStatus := 'Sequence failed'; END_IF
            IF _stLastResult.bHasError THEN
                stLastError := _stLastResult.stError;
                // Single audit-trail bridge: surface the runtime result error to the global logger.
                GVL_ErrorLogger.Logger.LogError(
                    sSource        := stLastError.sSource,
                    eErrorId       := stLastError.eErrorId,
                    sContext       := stLastError.sMessage,
                    eSeverity      := stLastError.eSeverity,
                    fCurrentValue  := stLastError.fCurrentValue,
                    fExpectedValue := stLastError.fExpectedValue,
                    sUnits         := stLastError.sUnits);
            END_IF
            // Drive hardware to a safe state on failure (Halt cascades to all child nodes).
            IF _ipActiveSequence <> 0 THEN
                _ipActiveSequence.Halt();
            END_IF
            eActiveSequence := E_Sequence.Error;
            bBusy           := FALSE;
            bError          := TRUE;
    END_CASE
END_METHOD

METHOD PRIVATE _MapSide : BOOL
VAR_INPUT
    nSide : INT;
END_VAR
VAR_OUTPUT
    eSide : E_GasSide;
END_VAR
    CASE nSide OF
        1: eSide := E_GasSide.A_SIDE;
        2: eSide := E_GasSide.B_SIDE;
    ELSE
        sStatus := 'Invalid side';
        RETURN;
    END_CASE
    _MapSide := TRUE;
END_METHOD

METHOD PRIVATE _AbortCurrentSequence
    IF _ipActiveSequence <> 0 THEN
        _ipActiveSequence.Halt();   // drive owned hardware to safe state, freeze logic
        _ipActiveSequence.Reset();  // rewind so the sequence can run again
    END_IF
END_METHOD

METHOD PRIVATE _SetError
VAR_INPUT
    sMsg : STRING(255);
    eErrorId : E_ErrorId := E_ErrorId.ERR_GEN_INITIALIZATION;
END_VAR
    // Drive hardware to a safe state before abandoning the active sequence.
    IF _ipActiveSequence <> 0 THEN
        _ipActiveSequence.Halt();
    END_IF
    sStatus                       := sMsg;
    eActiveSequence               := E_Sequence.Error;
    _ipActiveSequence             := 0;
    bError                        := TRUE;
    bBusy                         := FALSE;
    bDone                         := FALSE;
    stLastError.eErrorId          := eErrorId;
    stLastError.eSeverity         := E_TcEventSeverity.Error;
    stLastError.sSource           := 'FB_SequenceOrchestrator';
    stLastError.sMessage          := sMsg;
    stLastError.tTimestamp        := F_GetCurrentDT();
    stLastError.tOriginTimestamp  := stLastError.tTimestamp;
END_METHOD

METHOD PRIVATE _CompleteSequence
    sStatus         := 'Completed';
    eActiveSequence := E_Sequence.None;
    _ipActiveSequence := 0;
    bBusy           := FALSE;
    bDone           := TRUE;
    bError          := FALSE;
    rProgress       := 100.0;
END_METHOD

METHOD PRIVATE _ResetState
    IF _ipActiveSequence <> 0 THEN
        _ipActiveSequence.Reset();
    END_IF
    eActiveSequence   := E_Sequence.None;
    _ipActiveSequence := 0;
    bBusy             := FALSE;
    bDone             := FALSE;
    bError            := FALSE;
    rProgress         := 0.0;
    MEMSET(ADR(stLastError), 0, SIZEOF(stLastError));
    sStatus           := 'Ready';
END_METHOD

METHOD PRIVATE _UpdateLastPurgedBubbler
    IF eActiveSequence = E_Sequence.PurgePrecursor OR eActiveSequence = E_Sequence.PurgeReactant THEN
        IF _nBubblerIndex > 0 THEN
            IF _eSide = E_GasSide.A_SIDE THEN
                nLastPurgedBubblerA := DINT_TO_INT(_nBubblerIndex);
            ELSE
                nLastPurgedBubblerB := DINT_TO_INT(_nBubblerIndex);
            END_IF
        END_IF
    END_IF
END_METHOD

METHOD PRIVATE _InitiateSystemStop : BOOL
VAR_INPUT
    sLabel : STRING(255);
END_VAR
    _AbortCurrentSequence();
    _ResetState();

    IF NOT _fbSystemStop.Init(ipProvider := _ipProvider) THEN
        _SetError(CONCAT(sLabel, ' init failed'));
        RETURN;
    END_IF
    _ipActiveSequence    := _fbSystemStop;
    _Start(E_Sequence.Stop, CONCAT(sLabel, '...'));
    _InitiateSystemStop  := TRUE;
END_METHOD
